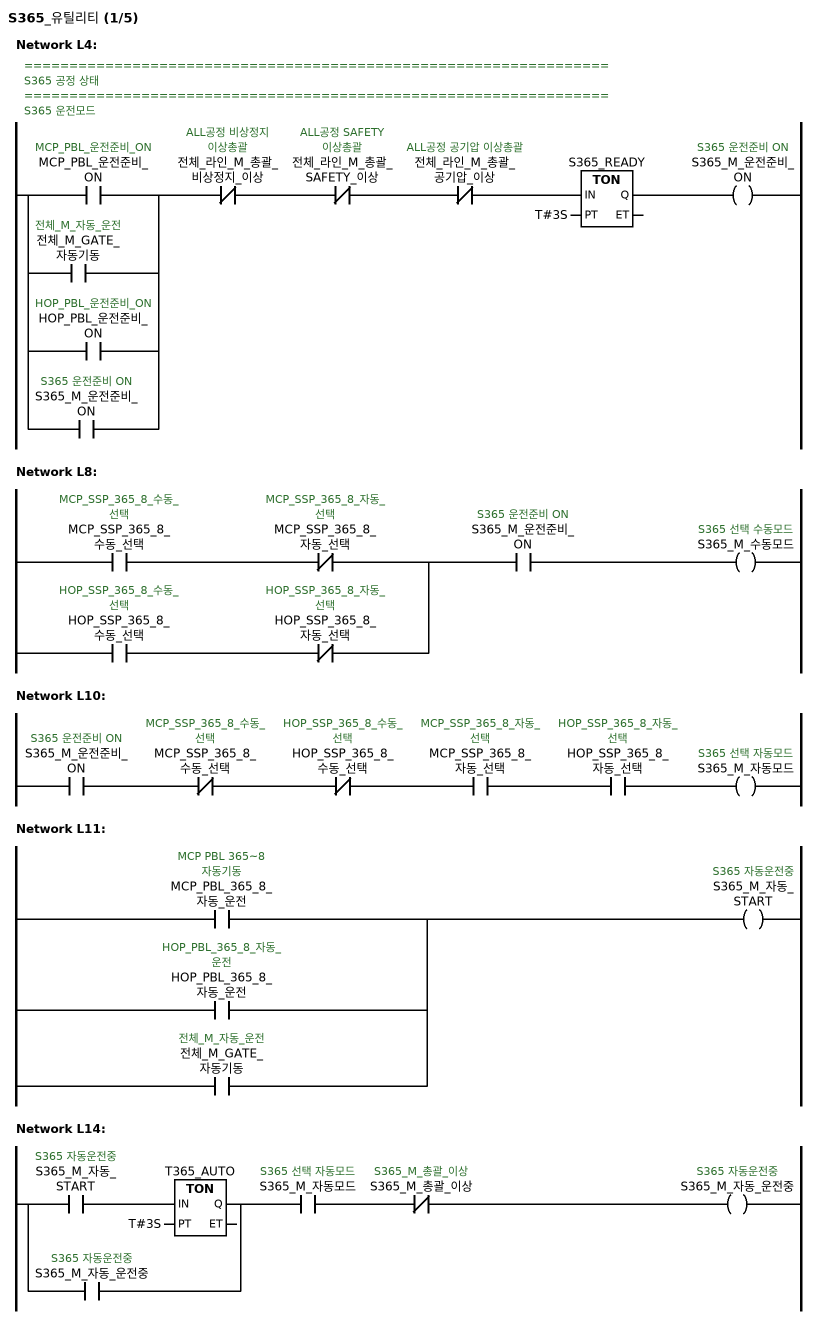
(* [picture p168: S365_유틸리티 rungs L4-L14] *)
(* ================================================================= *)
(* S365 공정 상태 *)
(* ================================================================= *)
(* S365 운전모드 *)
(* Rung L4 *)
S365_READY(IN := (MCP_PBL_운전준비_ON OR 전체_M_GATE_자동기동 OR HOP_PBL_운전준비_ON OR S365_M_운전준비_ON) AND NOT 전체_라인_M_총괄_비상정지_이상 AND NOT 전체_라인_M_총괄_SAFETY_이상 AND NOT 전체_라인_M_총괄_공기압_이상, PT := T#3S);
S365_M_운전준비_ON := S365_READY.Q;
(* Rung L8 *)
S365_M_수동모드 := ((MCP_SSP_365_8_수동_선택 AND NOT MCP_SSP_365_8_자동_선택) OR (HOP_SSP_365_8_수동_선택 AND NOT HOP_SSP_365_8_자동_선택)) AND S365_M_운전준비_ON;
(* Rung L10 *)
S365_M_자동모드 := S365_M_운전준비_ON AND NOT MCP_SSP_365_8_수동_선택 AND NOT HOP_SSP_365_8_수동_선택 AND MCP_SSP_365_8_자동_선택 AND HOP_SSP_365_8_자동_선택;
(* Rung L11 *)
S365_M_자동_START := MCP_PBL_365_8_자동_운전 OR HOP_PBL_365_8_자동_운전 OR 전체_M_GATE_자동기동;
(* Rung L14 *)
T365_AUTO(IN := S365_M_자동_START, PT := T#3S);
S365_M_자동_운전중 := (T365_AUTO.Q OR S365_M_자동_운전중) AND S365_M_자동모드 AND NOT S365_M_총괄_이상;

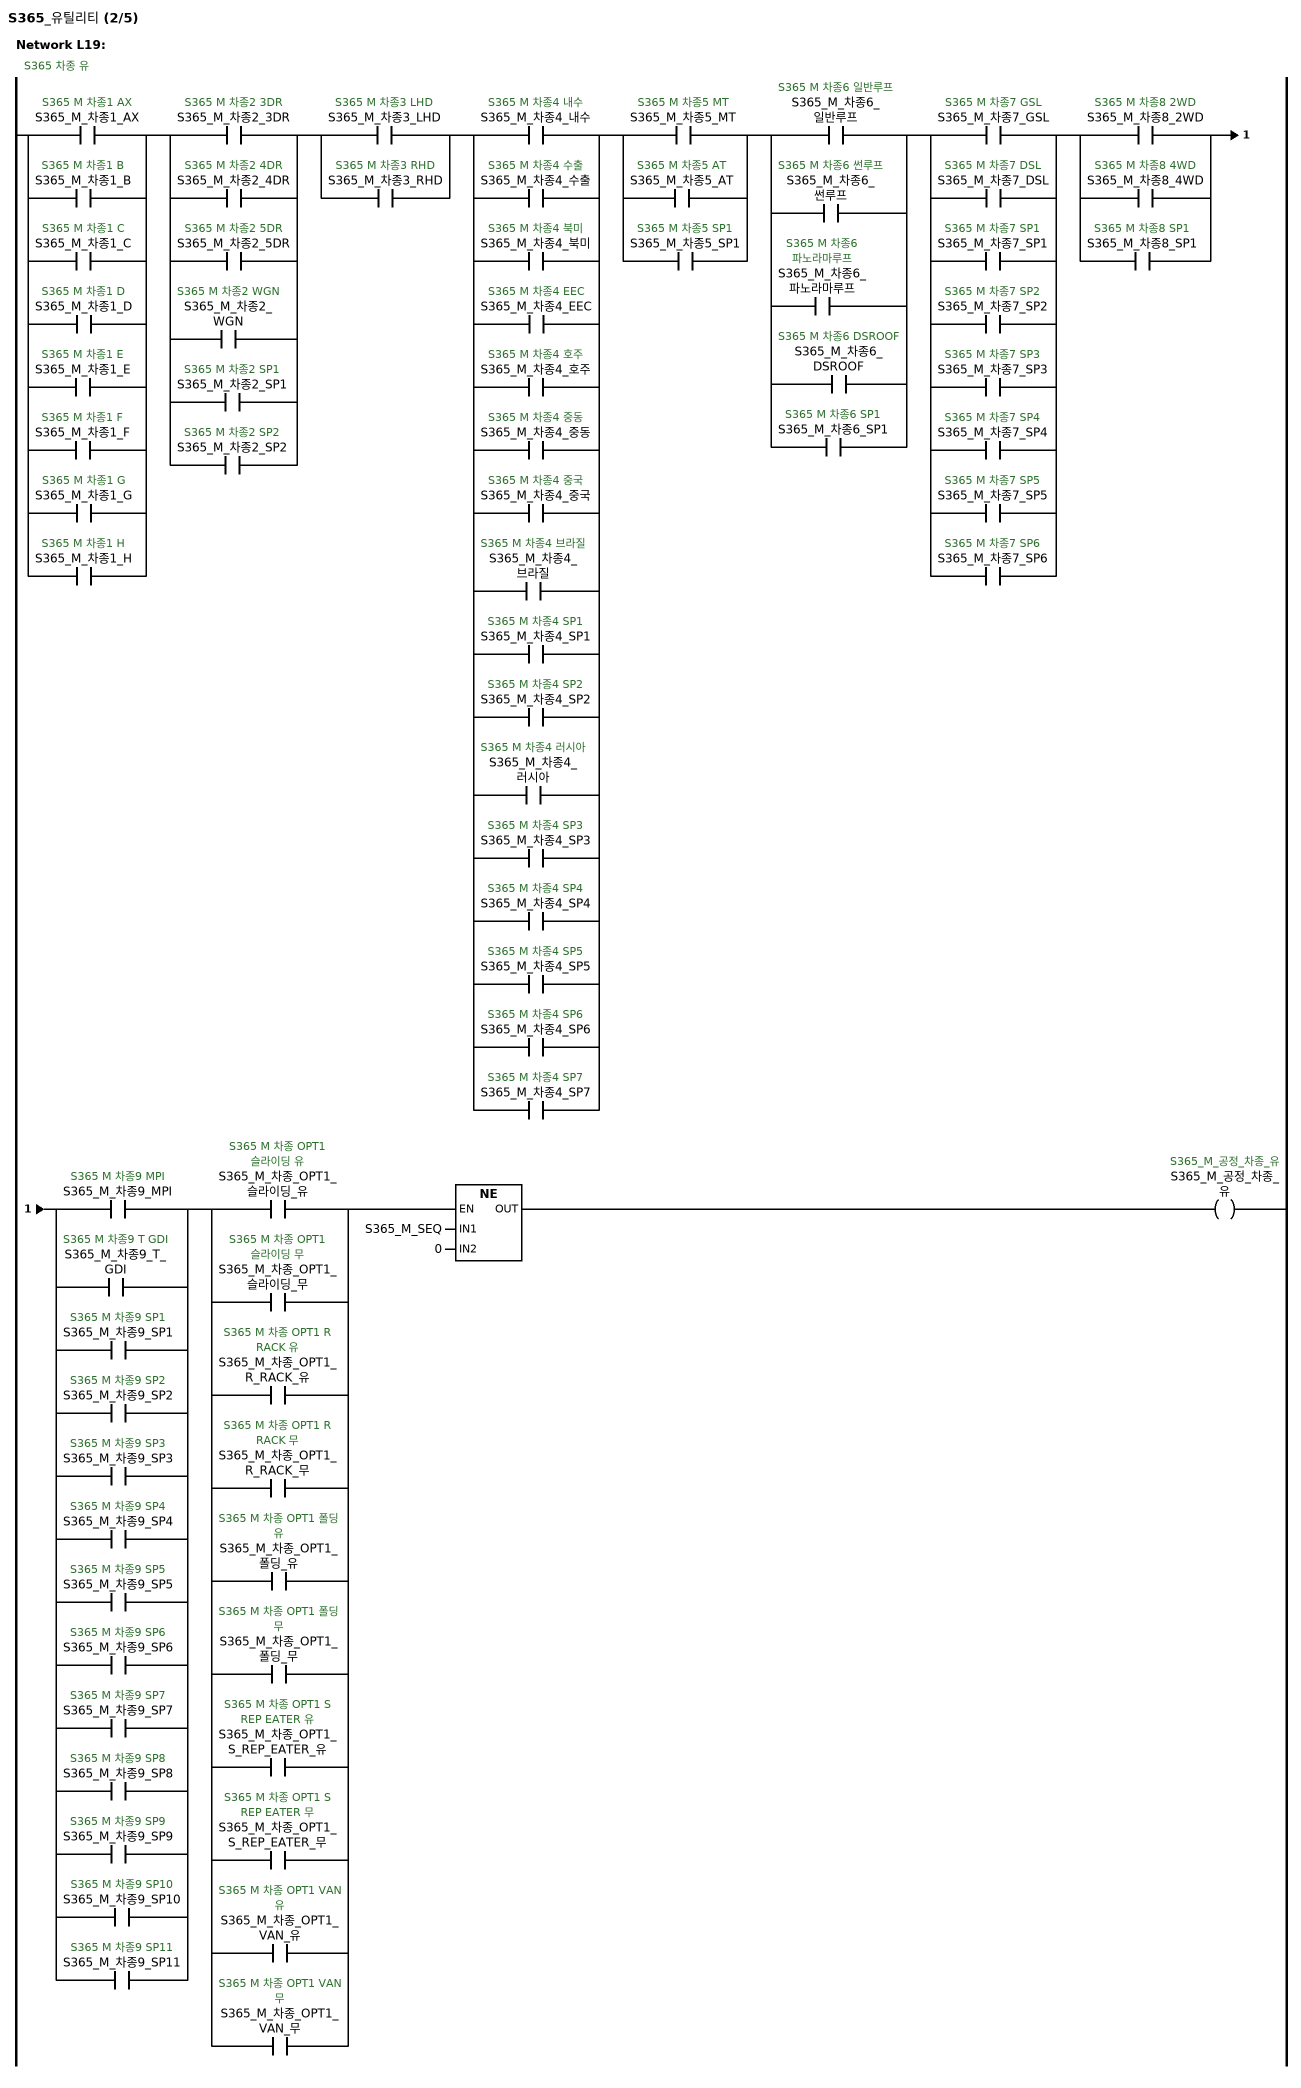
(* S365 차종 유 *)
(* Rung L19 *)
IF (S365_M_차종1_AX OR S365_M_차종1_B OR S365_M_차종1_C OR S365_M_차종1_D OR S365_M_차종1_E OR S365_M_차종1_F OR S365_M_차종1_G OR S365_M_차종1_H) AND (S365_M_차종2_3DR OR S365_M_차종2_4DR OR S365_M_차종2_5DR OR S365_M_차종2_WGN OR S365_M_차종2_SP1 OR S365_M_차종2_SP2) AND (S365_M_차종3_LHD OR S365_M_차종3_RHD) AND (S365_M_차종4_내수 OR S365_M_차종4_수출 OR S365_M_차종4_북미 OR S365_M_차종4_EEC OR S365_M_차종4_호주 OR S365_M_차종4_중동 OR S365_M_차종4_중국 OR S365_M_차종4_브라질 OR S365_M_차종4_SP1 OR S365_M_차종4_SP2 OR S365_M_차종4_러시아 OR S365_M_차종4_SP3 OR S365_M_차종4_SP4 OR S365_M_차종4_SP5 OR S365_M_차종4_SP6 OR S365_M_차종4_SP7) AND (S365_M_차종5_MT OR S365_M_차종5_AT OR S365_M_차종5_SP1) AND (S365_M_차종6_일반루프 OR S365_M_차종6_썬루프 OR S365_M_차종6_파노라마루프 OR S365_M_차종6_DSROOF OR S365_M_차종6_SP1) AND (S365_M_차종7_GSL OR S365_M_차종7_DSL OR S365_M_차종7_SP1 OR S365_M_차종7_SP2 OR S365_M_차종7_SP3 OR S365_M_차종7_SP4 OR S365_M_차종7_SP5 OR S365_M_차종7_SP6) AND (S365_M_차종8_2WD OR S365_M_차종8_4WD OR S365_M_차종8_SP1) AND (S365_M_차종9_MPI OR S365_M_차종9_T_GDI OR S365_M_차종9_SP1 OR S365_M_차종9_SP2 OR S365_M_차종9_SP3 OR S365_M_차종9_SP4 OR S365_M_차종9_SP5 OR S365_M_차종9_SP6 OR S365_M_차종9_SP7 OR S365_M_차종9_SP8 OR S365_M_차종9_SP9 OR S365_M_차종9_SP10 OR S365_M_차종9_SP11) AND (S365_M_차종_OPT1_슬라이딩_유 OR S365_M_차종_OPT1_슬라이딩_무 OR S365_M_차종_OPT1_R_RACK_유 OR S365_M_차종_OPT1_R_RACK_무 OR S365_M_차종_OPT1_폴딩_유 OR S365_M_차종_OPT1_폴딩_무 OR S365_M_차종_OPT1_S_REP_EATER_유 OR S365_M_차종_OPT1_S_REP_EATER_무 OR S365_M_차종_OPT1_VAN_유 OR S365_M_차종_OPT1_VAN_무) THEN
    _t1 := S365_M_SEQ <> 0;
END_IF;
S365_M_공정_차종_유 := _t1;

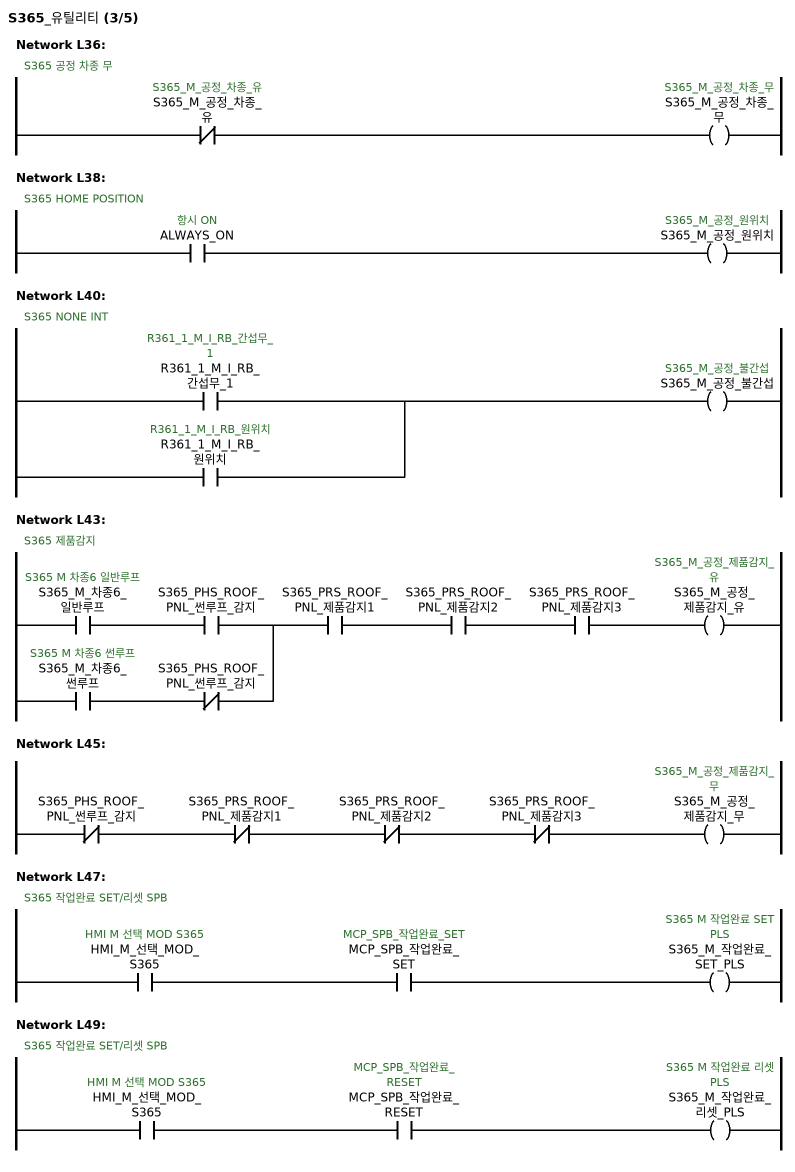
(* S365 공정 차종 무 *)
(* Rung L36 *)
S365_M_공정_차종_무 := NOT S365_M_공정_차종_유;
(* S365 HOME POSITION *)
(* Rung L38 *)
S365_M_공정_원위치 := ALWAYS_ON;
(* S365 NONE INT *)
(* Rung L40 *)
S365_M_공정_불간섭 := R361_1_M_I_RB_간섭무_1 OR R361_1_M_I_RB_원위치;
(* S365 제품감지 *)
(* Rung L43 *)
S365_M_공정_제품감지_유 := ((S365_M_차종6_일반루프 AND S365_PHS_ROOF_PNL_썬루프_감지) OR (S365_M_차종6_썬루프 AND NOT S365_PHS_ROOF_PNL_썬루프_감지)) AND S365_PRS_ROOF_PNL_제품감지1 AND S365_PRS_ROOF_PNL_제품감지2 AND S365_PRS_ROOF_PNL_제품감지3;
(* Rung L45 *)
S365_M_공정_제품감지_무 := NOT S365_PHS_ROOF_PNL_썬루프_감지 AND NOT S365_PRS_ROOF_PNL_제품감지1 AND NOT S365_PRS_ROOF_PNL_제품감지2 AND NOT S365_PRS_ROOF_PNL_제품감지3;
(* S365 작업완료 SET/리셋 SPB *)
(* Rung L47 *)
S365_M_작업완료_SET_PLS := HMI_M_선택_MOD_S365 AND MCP_SPB_작업완료_SET;
(* S365 작업완료 SET/리셋 SPB *)
(* Rung L49 *)
S365_M_작업완료_리셋_PLS := HMI_M_선택_MOD_S365 AND MCP_SPB_작업완료_RESET;

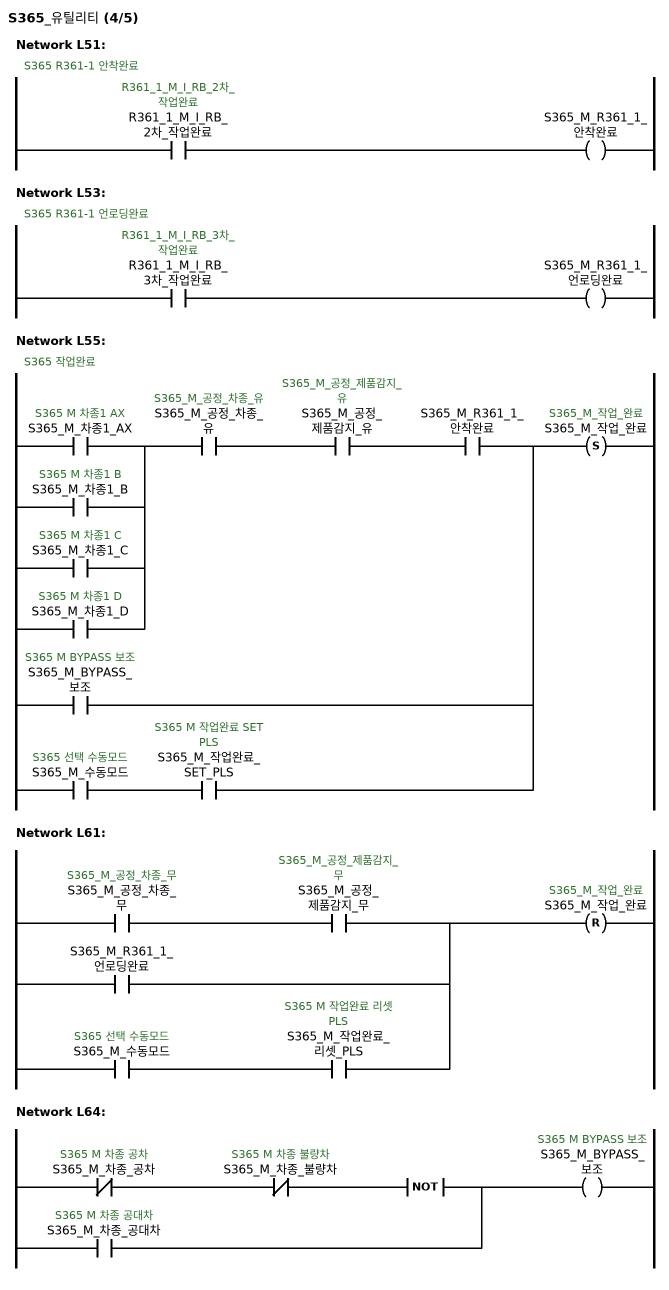
(* S365 R361-1 안착완료 *)
(* Rung L51 *)
S365_M_R361_1_안착완료 := R361_1_M_I_RB_2차_작업완료;
(* S365 R361-1 언로딩완료 *)
(* Rung L53 *)
S365_M_R361_1_언로딩완료 := R361_1_M_I_RB_3차_작업완료;
(* S365 작업완료 *)
(* Rung L55 *)
IF ((S365_M_차종1_AX OR S365_M_차종1_B OR S365_M_차종1_C OR S365_M_차종1_D) AND S365_M_공정_차종_유 AND S365_M_공정_제품감지_유 AND S365_M_R361_1_안착완료) OR S365_M_BYPASS_보조 OR (S365_M_수동모드 AND S365_M_작업완료_SET_PLS) THEN
    S365_M_작업_완료 := TRUE;
END_IF;
(* Rung L61 *)
IF (S365_M_공정_차종_무 AND S365_M_공정_제품감지_무) OR S365_M_R361_1_언로딩완료 OR (S365_M_수동모드 AND S365_M_작업완료_리셋_PLS) THEN
    S365_M_작업_완료 := FALSE;
END_IF;
(* Rung L64 *)
S365_M_BYPASS_보조 := NOT (NOT S365_M_차종_공차 AND NOT S365_M_차종_불량차) OR S365_M_차종_공대차;

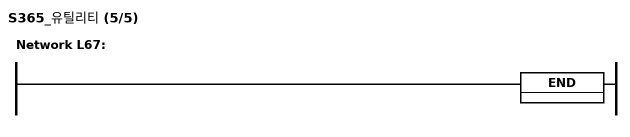
(* Rung L67 *)
END();
END_PROGRAM

PROGRAM S365_이상 (* task: 스캔 프로그램 *)
VAR
    INST10 : TON;
    INST11 : TON;
    INST12 : TON;
    INST13 : TON;
    INST14 : TON;
    INST15 : TON;
    INST16 : TON;
    INST17 : TON;
    INST18 : TON;
    INST19 : TON;
    INST20 : TON;
    INST21 : TON;
    INST22 : TON;
    INST23 : TON;
    INST24 : TON;
    INST25 : TON;
    INST8 : TON;
    INST9 : TON;
END_VAR
VAR_EXTERNAL RETAIN
    S362_M_자동_운전중 : BOOL; (* AT %MW1000.4 *) (* S362 자동운전중 *)
    S365_M_NODE_6_01_통신_이상 : BOOL; (* AT %MW2524.0 *)
    S365_M_R361_1_안착완료 : BOOL; (* AT %MW2501.1 *)
    S365_M_공정_불간섭 : BOOL; (* AT %MW2504.1 *) (* S365_M_공정_불간섭 *)
    S365_M_공정_제품감지_무 : BOOL; (* AT %MW2501.4 *) (* S365_M_공정_제품감지_무 *)
    S365_M_공정_제품감지_유 : BOOL; (* AT %MW2501.3 *) (* S365_M_공정_제품감지_유 *)
    S365_M_공정_차종_유 : BOOL; (* AT %MW2502.0 *) (* S365_M_공정_차종_유 *)
    S365_M_자동_운전중 : BOOL; (* AT %MW2500.4 *) (* S365 자동운전중 *)
    S365_M_차종6_썬루프 : BOOL; (* AT %MW10143.4 *) (* S365 M 차종6 썬루프 *)
    S365_M_차종6_일반루프 : BOOL; (* AT %MW10143.3 *) (* S365 M 차종6 일반루프 *)
    S365_M_총괄_CP_이상 : BOOL; (* AT %MW2509.7 *) (* S365 CP OFF 이상 *)
    S365_M_총괄_CT_이상 : BOOL; (* AT %MW2510.4 *) (* S365   TACK TIME 이상 *)
    S365_M_총괄_EOCR_이상 : BOOL; (* AT %MW2509.8 *) (* S365_M_총괄_EOCR_이상 *)
    S365_M_총괄_INV_이상 : BOOL; (* AT %MW2509.9 *) (* S365_M_총괄_INV_이상 *)
    S365_M_총괄_LS_이상 : BOOL; (* AT %MW2509.15 *) (* S365 LS 이상 *)
    S365_M_총괄_MATCH_이상 : BOOL; (* AT %MW2510.0 *) (* S365 매트SW 이상 *)
    S365_M_총괄_MC_이상 : BOOL; (* AT %MW2509.13 *) (* S365_M_총괄_MC_이상 *)
    S365_M_총괄_NFB_이상 : BOOL; (* AT %MW2509.11 *) (* S365_M_총괄_NFB_이상 *)
    S365_M_총괄_ROBOT_이상 : BOOL; (* AT %MW2510.1 *) (* S365 ROBOT 이상 *)
    S365_M_총괄_SAFETY_이상 : BOOL; (* AT %MW2509.2 *) (* S365 SAFETY 이상 *)
    S365_M_총괄_공기압_이상 : BOOL; (* AT %MW2509.3 *) (* S365 공기압 이상 *)
    S365_M_총괄_사양_이상 : BOOL; (* AT %MW2509.6 *) (* S365 사양 이상 *)
    S365_M_총괄_오버런_이상 : BOOL; (* AT %MW2509.12 *) (* S365_M_총괄_오버런_이상 *)
    S365_M_총괄_용접타점수_이상 : BOOL; (* AT %MW2510.2 *) (* S365 용접타점수 이상 *)
    S365_M_총괄_이상 : BOOL; (* AT %MW2509.0 *) (* S365_M_총괄_이상 *)
    S365_M_총괄_제품감지_이상 : BOOL; (* AT %MW2509.4 *) (* S365 제품감지 이상 *)
    S365_M_총괄_차종_이상 : BOOL; (* AT %MW2509.5 *) (* S365 차종 이상 *)
    S365_M_총괄_통신_이상 : BOOL; (* AT %MW2509.14 *) (* S365 통신이상 *)
    전체_M_이상_리셋 : BOOL; (* AT %MW308.2 *) (* ALL공정 PB 이상리셋 *)
END_VAR
VAR_EXTERNAL
    S365_6_1_PLC_BOX_CP_TRIP : BOOL; (* AT %MW86012.15 *) (* S365_6_1_PLC_BOX_CP_TRIP *)
    S365_PHS_ROOF_PNL_썬루프_감지 : BOOL; (* AT %MW86010.3 *)
    _0006_EB01_CFG_ER : BOOL; (* AT %MW186022.0 *) (* EB 구성 에러 *)
    _0006_EB01_DEER : BOOL; (* AT %MW186022.1 *) (* EB 운전 중 탈락 *)
    _0006_EB01_IO_DEER : BOOL; (* AT %MW186023.2 *) (* EB IO 탈락 에러 *)
    _0006_EB01_IO_TYER : BOOL; (* AT %MW186023.1 *) (* EB IO 타입 에러 *)
    _0007_EB10_CFG_ER : BOOL; (* AT %MW187040.0 *) (* EB 구성 에러 *)
    _0007_EB10_DEER : BOOL; (* AT %MW187040.1 *) (* EB 운전 중 탈락 *)
    _0007_EB10_IO_DEER : BOOL; (* AT %MW187041.2 *) (* EB IO 탈락 에러 *)
    _0007_EB10_IO_TYER : BOOL; (* AT %MW187041.1 *) (* EB IO 타입 에러 *)
END_VAR

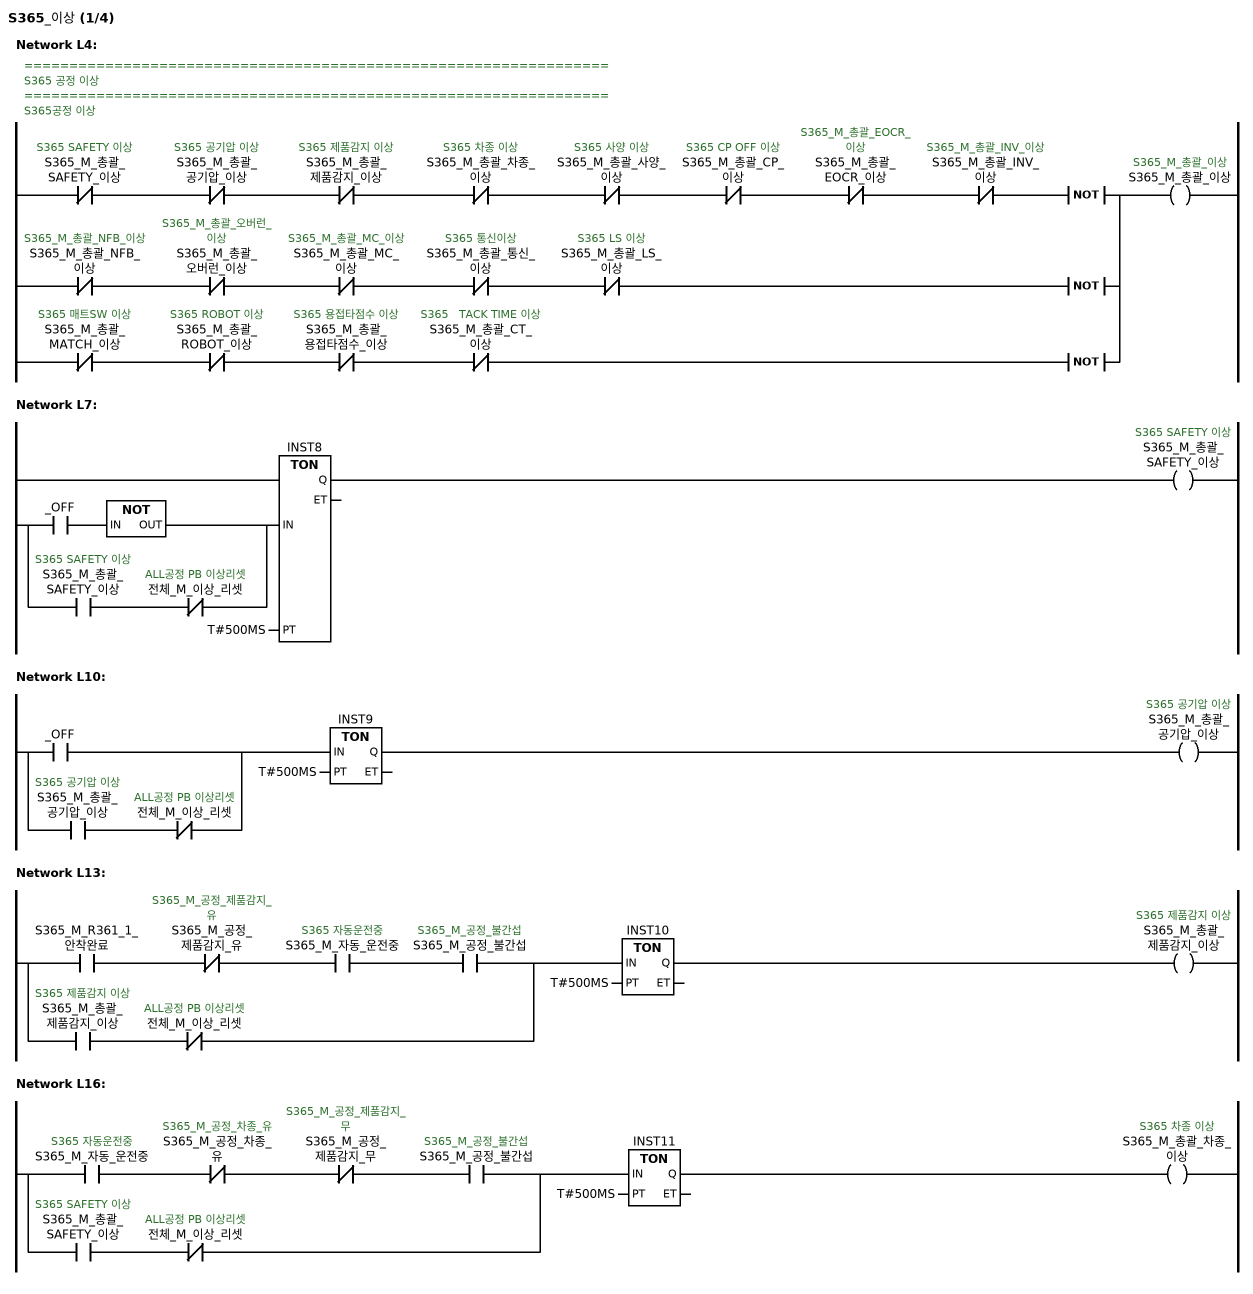
(* ================================================================= *)
(* S365 공정 이상 *)
(* ================================================================= *)
(* S365공정 이상 *)
(* Rung L4 *)
S365_M_총괄_이상 := NOT (NOT S365_M_총괄_SAFETY_이상 AND NOT S365_M_총괄_공기압_이상 AND NOT S365_M_총괄_제품감지_이상 AND NOT S365_M_총괄_차종_이상 AND NOT S365_M_총괄_사양_이상 AND NOT S365_M_총괄_CP_이상 AND NOT S365_M_총괄_EOCR_이상 AND NOT S365_M_총괄_INV_이상) OR NOT (NOT S365_M_총괄_NFB_이상 AND NOT S365_M_총괄_오버런_이상 AND NOT S365_M_총괄_MC_이상 AND NOT S365_M_총괄_통신_이상 AND NOT S365_M_총괄_LS_이상) OR NOT (NOT S365_M_총괄_MATCH_이상 AND NOT S365_M_총괄_ROBOT_이상 AND NOT S365_M_총괄_용접타점수_이상 AND NOT S365_M_총괄_CT_이상);
(* Rung L7 *)
INST8(IN := (NOT _OFF) OR (S365_M_총괄_SAFETY_이상 AND NOT 전체_M_이상_리셋), PT := T#500MS);
S365_M_총괄_SAFETY_이상 := INST8.Q;
(* Rung L10 *)
INST9(IN := _OFF OR (S365_M_총괄_공기압_이상 AND NOT 전체_M_이상_리셋), PT := T#500MS);
S365_M_총괄_공기압_이상 := INST9.Q;
(* Rung L13 *)
INST10(IN := (S365_M_R361_1_안착완료 AND NOT S365_M_공정_제품감지_유 AND S365_M_자동_운전중 AND S365_M_공정_불간섭) OR (S365_M_총괄_제품감지_이상 AND NOT 전체_M_이상_리셋), PT := T#500MS);
S365_M_총괄_제품감지_이상 := INST10.Q;
(* Rung L16 *)
INST11(IN := (S365_M_자동_운전중 AND NOT S365_M_공정_차종_유 AND NOT S365_M_공정_제품감지_무 AND S365_M_공정_불간섭) OR (S365_M_총괄_SAFETY_이상 AND NOT 전체_M_이상_리셋), PT := T#500MS);
S365_M_총괄_차종_이상 := INST11.Q;

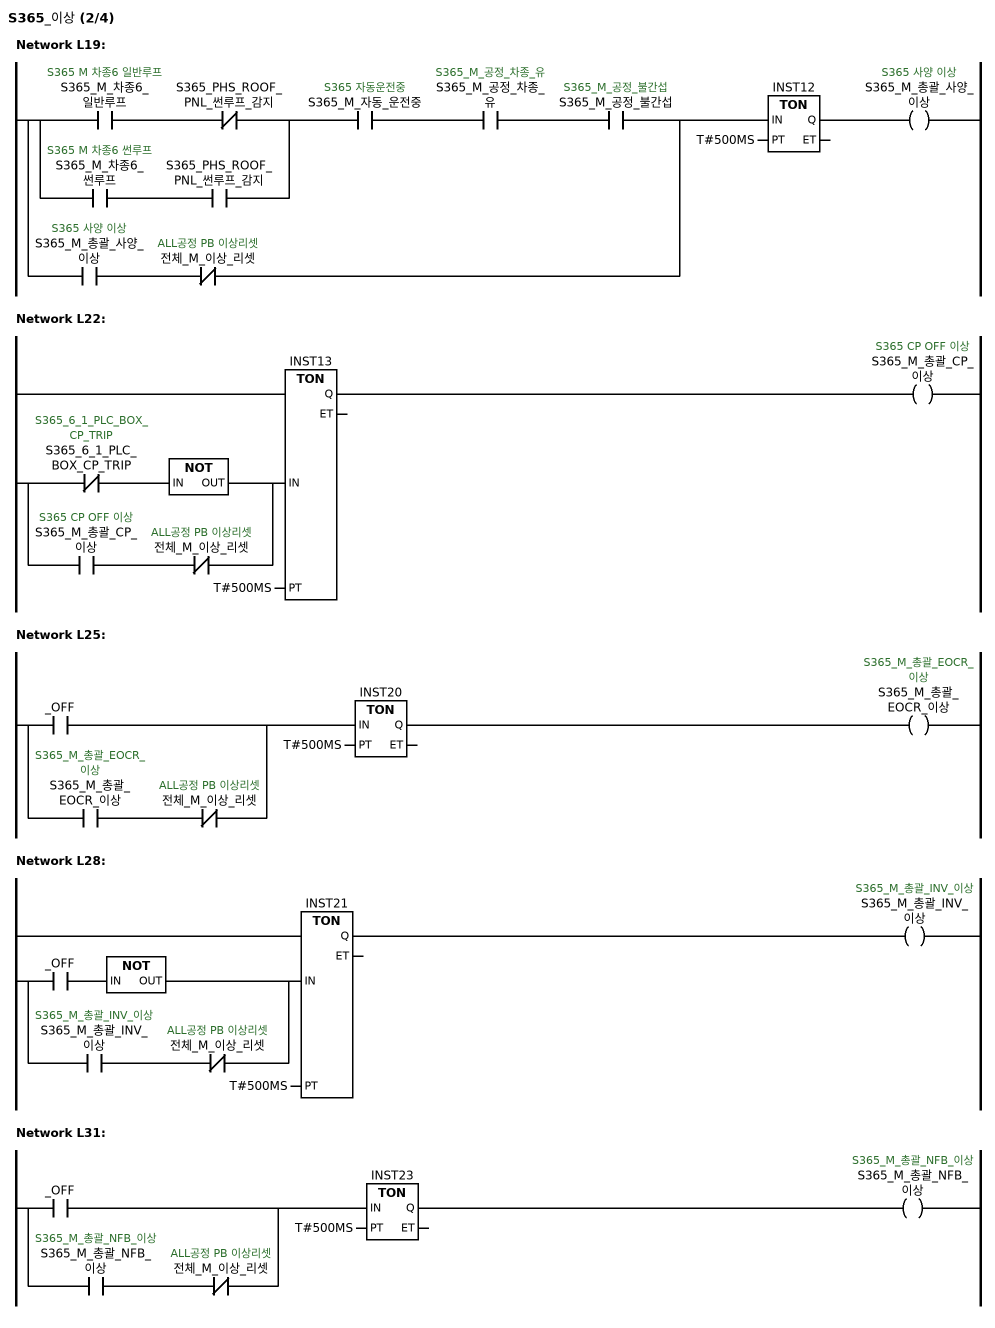
(* Rung L19 *)
INST12(IN := (((S365_M_차종6_일반루프 AND NOT S365_PHS_ROOF_PNL_썬루프_감지) OR (S365_M_차종6_썬루프 AND S365_PHS_ROOF_PNL_썬루프_감지)) AND S365_M_자동_운전중 AND S365_M_공정_차종_유 AND S365_M_공정_불간섭) OR (S365_M_총괄_사양_이상 AND NOT 전체_M_이상_리셋), PT := T#500MS);
S365_M_총괄_사양_이상 := INST12.Q;
(* Rung L22 *)
INST13(IN := (NOT (NOT S365_6_1_PLC_BOX_CP_TRIP)) OR (S365_M_총괄_CP_이상 AND NOT 전체_M_이상_리셋), PT := T#500MS);
S365_M_총괄_CP_이상 := INST13.Q;
(* Rung L25 *)
INST20(IN := _OFF OR (S365_M_총괄_EOCR_이상 AND NOT 전체_M_이상_리셋), PT := T#500MS);
S365_M_총괄_EOCR_이상 := INST20.Q;
(* Rung L28 *)
INST21(IN := (NOT _OFF) OR (S365_M_총괄_INV_이상 AND NOT 전체_M_이상_리셋), PT := T#500MS);
S365_M_총괄_INV_이상 := INST21.Q;
(* Rung L31 *)
INST23(IN := _OFF OR (S365_M_총괄_NFB_이상 AND NOT 전체_M_이상_리셋), PT := T#500MS);
S365_M_총괄_NFB_이상 := INST23.Q;

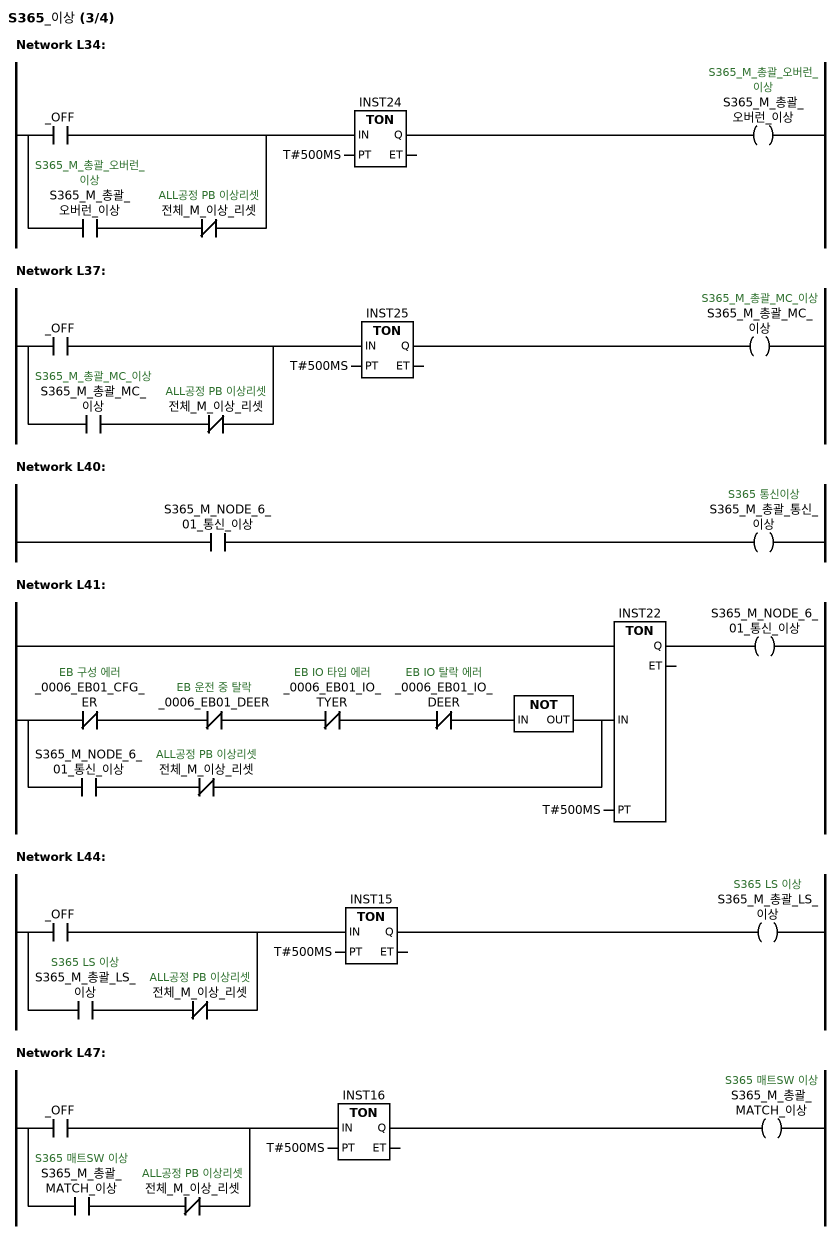
(* Rung L34 *)
INST24(IN := _OFF OR (S365_M_총괄_오버런_이상 AND NOT 전체_M_이상_리셋), PT := T#500MS);
S365_M_총괄_오버런_이상 := INST24.Q;
(* Rung L37 *)
INST25(IN := _OFF OR (S365_M_총괄_MC_이상 AND NOT 전체_M_이상_리셋), PT := T#500MS);
S365_M_총괄_MC_이상 := INST25.Q;
(* Rung L40 *)
S365_M_총괄_통신_이상 := S365_M_NODE_6_01_통신_이상;
(* Rung L41 *)
INST22(IN := (NOT (NOT _0006_EB01_CFG_ER AND NOT _0006_EB01_DEER AND NOT _0006_EB01_IO_TYER AND NOT _0006_EB01_IO_DEER)) OR (S365_M_NODE_6_01_통신_이상 AND NOT 전체_M_이상_리셋), PT := T#500MS);
S365_M_NODE_6_01_통신_이상 := INST22.Q;
(* Rung L44 *)
INST15(IN := _OFF OR (S365_M_총괄_LS_이상 AND NOT 전체_M_이상_리셋), PT := T#500MS);
S365_M_총괄_LS_이상 := INST15.Q;
(* Rung L47 *)
INST16(IN := _OFF OR (S365_M_총괄_MATCH_이상 AND NOT 전체_M_이상_리셋), PT := T#500MS);
S365_M_총괄_MATCH_이상 := INST16.Q;

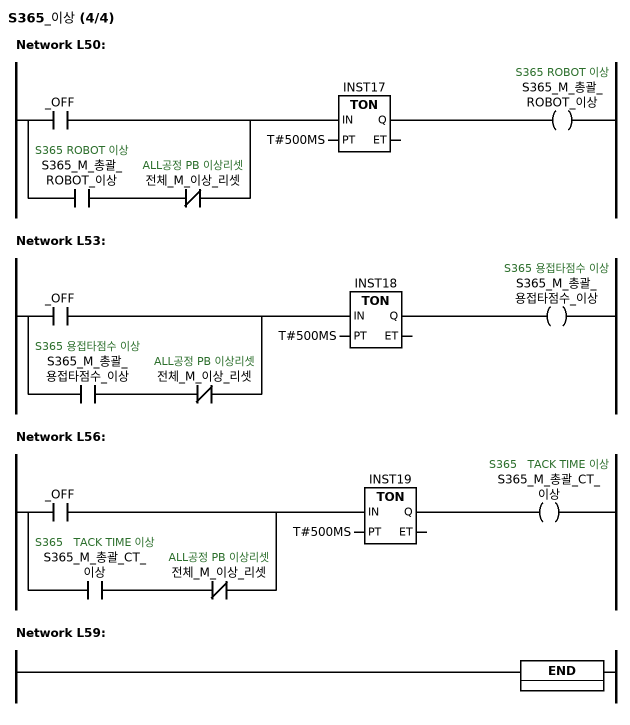
(* Rung L50 *)
INST17(IN := _OFF OR (S365_M_총괄_ROBOT_이상 AND NOT 전체_M_이상_리셋), PT := T#500MS);
S365_M_총괄_ROBOT_이상 := INST17.Q;
(* Rung L53 *)
INST18(IN := _OFF OR (S365_M_총괄_용접타점수_이상 AND NOT 전체_M_이상_리셋), PT := T#500MS);
S365_M_총괄_용접타점수_이상 := INST18.Q;
(* Rung L56 *)
INST19(IN := _OFF OR (S365_M_총괄_CT_이상 AND NOT 전체_M_이상_리셋), PT := T#500MS);
S365_M_총괄_CT_이상 := INST19.Q;
(* Rung L59 *)
END();
END_PROGRAM

PROGRAM S366_유틸리티 (* task: 스캔 프로그램 *)
VAR
    A차종 : BOOL;
    C차종 : BOOL;
    S366_READY : TON;
    T365_AUTO : TON;
    WORK_1ST : BOOL;
END_VAR
VAR_EXTERNAL
    EGIS_CWS : BOOL;
    HOP_PBL_365_8_자동_운전 : BOOL; (* AT %MW87500.7 *) (* HOP_PBL_365_8_자동_운전 *)
    HOP_PBL_운전준비_ON : BOOL; (* AT %MW87500.0 *) (* HOP_PBL_운전준비_ON *)
    HOP_SSP_365_8_수동_선택 : BOOL; (* AT %MW87500.6 *) (* HOP_SSP_365_8_수동_선택 *)
    HOP_SSP_365_8_자동_선택 : BOOL; (* AT %MW87500.5 *) (* HOP_SSP_365_8_자동_선택 *)
    MCP_PBL_365_8_자동_운전 : BOOL; (* AT %MW87630.7 *) (* MCP PBL 365~8 자동기동 *)
    MCP_PBL_운전준비_ON : BOOL; (* AT %MW87630.0 *) (* MCP_PBL_운전준비_ON *)
    MCP_SPB_작업완료_RESET : BOOL; (* AT %MW87631.6 *) (* MCP_SPB_작업완료_RESET *)
    MCP_SPB_작업완료_SET : BOOL; (* AT %MW87631.7 *) (* MCP_SPB_작업완료_SET *)
    MCP_SSP_365_8_수동_선택 : BOOL; (* AT %MW87630.5 *) (* MCP_SSP_365_8_수동_선택 *)
    MCP_SSP_365_8_자동_선택 : BOOL; (* AT %MW87630.6 *) (* MCP_SSP_365_8_자동_선택 *)
    R361_1_M_I_RB_3차_작업완료 : BOOL; (* AT %MW20011.4 *) (* R361_1_M_I_RB_3차_작업완료 *)
    R361_1_M_I_RB_4차_작업완료 : BOOL; (* AT %MW20011.5 *) (* R361_1_M_I_RB_4차_작업완료 *)
    R361_1_M_I_RB_5차_작업완료 : BOOL; (* AT %MW20011.6 *) (* R361_1_M_I_RB_5차_작업완료 *)
    R361_1_M_I_RB_간섭무_1 : BOOL; (* AT %MW20012.0 *) (* R361_1_M_I_RB_간섭무_1 *)
    R361_1_M_I_RB_원위치 : BOOL; (* AT %MW20010.3 *) (* R361_1_M_I_RB_원위치 *)
    R363_1_M_I_RB_간섭무_1 : BOOL; (* AT %MW20032.0 *) (* R363_1_M_I_RB_간섭무_1 *)
    R363_1_M_I_RB_원위치 : BOOL; (* AT %MW20030.3 *) (* R363_1_M_I_RB_원위치 *)
    R363_2_M_I_RB_2차_작업완료 : BOOL; (* AT %MW20041.3 *) (* R363_2_M_I_RB_2차_작업완료 *)
    R363_2_M_I_RB_간섭무_1 : BOOL; (* AT %MW20042.0 *) (* R363_2_M_I_RB_간섭무_1 *)
    R363_2_M_I_RB_원위치 : BOOL; (* AT %MW20040.3 *) (* R363_2_M_I_RB_원위치 *)
    R364_1_M_I_RB_1차_작업완료 : BOOL; (* AT %MW20051.2 *) (* R364_1_M_I_RB_1차_작업완료 *)
    R366_1_M_I_RB_1차_작업완료 : BOOL; (* AT %MW20061.2 *) (* R366_1_M_I_RB_1차_작업완료 *)
    R366_1_M_I_RB_3차_작업완료 : BOOL; (* AT %MW20061.4 *) (* R366_1_M_I_RB_3차_작업완료 *)
    R366_1_M_I_RB_간섭무_1 : BOOL; (* AT %MW20062.0 *) (* R366_1_M_I_RB_간섭무_1 *)
    R366_1_M_I_RB_원위치 : BOOL; (* AT %MW20060.3 *) (* R366_1_M_I_RB_원위치 *)
    S362_6_INV3_SAFETY1_ON : BOOL; (* AT %MW95015.5 *) (* S362_6_INV3_SAFETY1_ON *)
    S362_6_INV3_SAFETY2_ON : BOOL; (* AT %MW95015.6 *) (* S362_6_INV3_SAFETY2_ON *)
    S362_6_INV3_이상_리셋 : BOOL; (* AT %MW95015.3 *) (* S362_6_INV3_이상_리셋 *)
    S362_6_INV4_SAFETY1_ON : BOOL; (* AT %MW95015.13 *) (* S362_6_INV4_SAFETY1_ON *)
    S362_6_INV4_SAFETY2_ON : BOOL; (* AT %MW95015.14 *) (* S362_6_INV4_SAFETY2_ON *)
    S362_6_INV4_이상_리셋 : BOOL; (* AT %MW95015.11 *) (* S362_6_INV4_이상_리셋 *)
    S366L_PRS_AX_COM_CHECK : BOOL; (* AT %MW88100.8 *) (* S366L_PRS_AX_COM_CHECK *)
    S366L_PRS_AX_GR_CHECK : BOOL; (* AT %MW88100.9 *) (* S366L_PRS_AX_GR_CHECK *)
    S366L_PRS_AX_RAIL_CHECK : BOOL; (* AT %MW88100.11 *) (* S366L_PRS_AX_RAIL_CHECK *)
    S366L_PRS_AX_ROOF_FRT_CHECK : BOOL; (* AT %MW88100.12 *) (* S366L_PRS_AX_ROOF_FRT_CHECK *)
    S366L_PRS_AX_ROOF_RR_CHECK : BOOL; (* AT %MW88100.13 *) (* S366L_PRS_AX_ROOF_RR_CHECK *)
    S366L_PRS_AX_SR_CHECK : BOOL; (* AT %MW88100.10 *) (* S366L_PRS_AX_SR_CHECK *)
    S366R_PRS_AX_COM_CHECK : BOOL; (* AT %MW88200.8 *) (* S366R_PRS_AX_COM_CHECK *)
    S366R_PRS_AX_GR_CHECK : BOOL; (* AT %MW88200.9 *) (* S366R_PRS_AX_GR_CHECK *)
    S366R_PRS_AX_RAIL_CHECK : BOOL; (* AT %MW88200.11 *) (* S366R_PRS_AX_RAIL_CHECK *)
    S366R_PRS_AX_ROOF_FRT_CHECK : BOOL; (* AT %MW88200.12 *) (* S366R_PRS_AX_ROOF_FRT_CHECK *)
    S366R_PRS_AX_ROOF_RR_CHECK : BOOL; (* AT %MW88200.13 *) (* S366R_PRS_AX_ROOF_RR_CHECK *)
    S366R_PRS_AX_SR_CHECK : BOOL; (* AT %MW88200.10 *) (* S366R_PRS_AX_SR_CHECK *)
    S366_LS_MAINTENANCE1 : BOOL; (* AT %MW86102.0 *)
    S366_LS_MAINTENANCE2 : BOOL; (* AT %MW86102.1 *)
END_VAR
VAR_EXTERNAL RETAIN
    HMI_M_선택_MOD_S364 : BOOL; (* AT %MW6.2 *) (* HMI M 선택 MOD S364 *)
    HMI_M_선택_MOD_S366 : BOOL; (* AT %MW6.4 *) (* HMI M 선택 MOD S366 *)
    R361_1_M_SEQ : WORD; (* AT %MW10000 *) (* R361 1 M SEQ *)
    R361_1_M_차종_유 : BOOL; (* AT %MW1502.0 *)
    S362_M_총괄_이상 : BOOL; (* AT %MW1009.0 *) (* S362_M_총괄_이상 *)
    S364_M_공정_차종_무 : BOOL; (* AT %MW2002.1 *) (* S364_M_공정_차종_무 *)
    S364_M_공정_차종_유 : BOOL; (* AT %MW2002.0 *) (* S364_M_공정_차종_유 *)
    S364_M_작업완료_SET_PLS : BOOL; (* AT %MW2000.8 *) (* S364 M 작업완료 SET PLS *)
    S364_M_작업완료_리셋_PLS : BOOL; (* AT %MW2000.9 *) (* S364 M 작업완료 리셋 PLS *)
    S366_M_AX_LH_CLP_전진단 : BOOL; (* AT %MW3104.3 *) (* S366_M_AX_LH_CLP_전진단 *)
    S366_M_AX_LH_CLP_후진단 : BOOL; (* AT %MW3104.4 *) (* S366_M_AX_LH_CLP_후진단 *)
    S366_M_AX_RH_CLP_전진단 : BOOL; (* AT %MW3112.3 *) (* S366_M_AX_RH_CLP_전진단 *)
    S366_M_AX_RH_CLP_후진단 : BOOL; (* AT %MW3112.4 *) (* S366_M_AX_RH_CLP_후진단 *)
    S366_M_BYPASS_보조 : BOOL; (* AT %MW3003.15 *) (* S366 M BYPASS 보조 *)
    S366_M_LH_TURN_1_포지션단 : BOOL; (* AT %MW3101.3 *) (* S366_M_LH_TURN_1_포지션단 *)
    S366_M_LH_TURN_2_포지션단 : BOOL; (* AT %MW3101.4 *) (* S366_M_LH_TURN_2_포지션단 *)
    S366_M_LH_TURN_3_포지션단 : BOOL; (* AT %MW3101.5 *) (* S366_M_LH_TURN_3_포지션단 *)
    S366_M_LH_TURN_4_포지션단 : BOOL; (* AT %MW3101.6 *) (* S366_M_LH_TURN_4_포지션단 *)
    S366_M_R361_1_ROOF_로딩완료 : BOOL; (* AT %MW3001.2 *)
    S366_M_R361_1_동일차종_OK : BOOL; (* AT %MW3005.8 *)
    S366_M_R361_1_언로딩완료 : BOOL; (* AT %MW3001.4 *)
    S366_M_R361_1_차종매칭_조건 : BOOL; (* AT %MW3005.0 *)
    S366_M_R363_2_RAIL_로딩완료 : BOOL; (* AT %MW3001.1 *)
    S366_M_R366_1_용접가능 : BOOL; (* AT %MW3004.10 *)
    S366_M_R366_1_용접완료 : BOOL; (* AT %MW3001.3 *)
    S366_M_RAIL_로딩가능 : BOOL; (* AT %MW3004.8 *)
    S366_M_RH_TURN_1_포지션단 : BOOL; (* AT %MW3109.3 *) (* S366_M_RH_TURN_1_포지션단 *)
    S366_M_RH_TURN_2_포지션단 : BOOL; (* AT %MW3109.4 *) (* S366_M_RH_TURN_2_포지션단 *)
    S366_M_RH_TURN_3_포지션단 : BOOL; (* AT %MW3109.5 *) (* S366_M_RH_TURN_3_포지션단 *)
    S366_M_RH_TURN_4_포지션단 : BOOL; (* AT %MW3109.6 *) (* S366_M_RH_TURN_4_포지션단 *)
    S366_M_ROOF_로딩가능 : BOOL; (* AT %MW3004.9 *)
    S366_M_SAFETY_불간섭 : BOOL; (* AT %MW3004.4 *) (* S366_M_SAFETY_불간섭 *)
    S366_M_SEQ : WORD; (* AT %MW10160 *) (* S366 M SEQ *)
    S366_M_TURN_LOCK_전진단 : BOOL; (* AT %MW3100.3 *) (* S366_M_TURN_LOCK_전진단 *)
    S366_M_TURN_LOCK_후진단 : BOOL; (* AT %MW3100.4 *) (* S366_M_TURN_LOCK_후진단 *)
    S366_M_공정_AX_FRT_PNL_제품감지_이상 : BOOL; (* AT %MW3014.4 *)
    S366_M_공정_FRT_PNL_제품감지_무 : BOOL; (* AT %MW3002.13 *)
    S366_M_공정_FRT_PNL_제품감지_유 : BOOL; (* AT %MW3002.12 *)
    S366_M_공정_RAIL_제품감지_무 : BOOL; (* AT %MW3001.15 *)
    S366_M_공정_RAIL_제품감지_유 : BOOL; (* AT %MW3001.14 *)
    S366_M_공정_RR_PNL_제품감지_무 : BOOL; (* AT %MW3002.15 *)
    S366_M_공정_RR_PNL_제품감지_유 : BOOL; (* AT %MW3002.14 *)
    S366_M_공정_공용_제품감지_무 : BOOL; (* AT %MW3001.9 *)
    S366_M_공정_공용_제품감지_유 : BOOL; (* AT %MW3001.8 *)
    S366_M_공정_불간섭 : BOOL; (* AT %MW3004.1 *) (* S366_M_공정_불간섭 *)
    S366_M_공정_썬루프_제품감지_무 : BOOL; (* AT %MW3001.13 *)
    S366_M_공정_썬루프_제품감지_유 : BOOL; (* AT %MW3001.12 *)
    S366_M_공정_원위치 : BOOL; (* AT %MW3004.0 *) (* S366_M_공정_원위치 *)
    S366_M_공정_일반루프_제품감지_무 : BOOL; (* AT %MW3001.11 *)
    S366_M_공정_일반루프_제품감지_유 : BOOL; (* AT %MW3001.10 *)
    S366_M_공정_제품감지_무 : BOOL; (* AT %MW3001.7 *) (* S366_M_공정_제품감지_무 *)
    S366_M_공정_제품감지_유 : BOOL; (* AT %MW3001.6 *) (* S366_M_공정_제품감지_유 *)
    S366_M_공정_차종_무 : BOOL; (* AT %MW3002.1 *) (* S366_M_공정_차종_무 *)
    S366_M_공정_차종_유 : BOOL; (* AT %MW3002.0 *) (* S366_M_공정_차종_유 *)
    S366_M_수동모드 : BOOL; (* AT %MW3000.3 *) (* S366 선택 수동모드 *)
    S366_M_운전준비_ON : BOOL; (* AT %MW3000.0 *) (* S366 운전준비 ON *)
    S366_M_자동_START : BOOL; (* AT %MW3000.5 *) (* S366 자동운전중 *)
    S366_M_자동_운전중 : BOOL; (* AT %MW3000.4 *) (* S366 자동운전중 *)
    S366_M_자동모드 : BOOL; (* AT %MW3000.1 *) (* S366 선택 자동모드 *)
    S366_M_작업_완료 : BOOL; (* AT %MW3001.0 *) (* S366_M_작업_완료 *)
    S366_M_작업완료_SET_PLS : BOOL; (* AT %MW3000.8 *) (* S366 M 작업완료 SET PLS *)
    S366_M_작업완료_리셋_PLS : BOOL; (* AT %MW3000.9 *) (* S366 M 작업완료 리셋 PLS *)
    S366_M_차종1_AX : BOOL; (* AT %MW10161.0 *) (* S366 M 차종1 AX *)
    S366_M_차종1_B : BOOL; (* AT %MW10161.1 *) (* S366 M 차종1 B *)
    S366_M_차종1_C : BOOL; (* AT %MW10161.2 *) (* S366 M 차종1 C *)
    S366_M_차종1_D : BOOL; (* AT %MW10161.3 *) (* S366 M 차종1 D *)
    S366_M_차종1_E : BOOL; (* AT %MW10161.4 *) (* S366 M 차종1 E *)
    S366_M_차종1_F : BOOL; (* AT %MW10161.5 *) (* S366 M 차종1 F *)
    S366_M_차종1_G : BOOL; (* AT %MW10161.6 *) (* S366 M 차종1 G *)
    S366_M_차종1_H : BOOL; (* AT %MW10161.7 *) (* S366 M 차종1 H *)
    S366_M_차종2_3DR : BOOL; (* AT %MW10161.8 *) (* S366 M 차종2 3DR *)
    S366_M_차종2_4DR : BOOL; (* AT %MW10161.9 *) (* S366 M 차종2 4DR *)
    S366_M_차종2_5DR : BOOL; (* AT %MW10161.10 *) (* S366 M 차종2 5DR *)
    S366_M_차종2_SP1 : BOOL; (* AT %MW10161.12 *) (* S366 M 차종2 SP1 *)
    S366_M_차종2_SP2 : BOOL; (* AT %MW10161.13 *) (* S366 M 차종2 SP2 *)
    S366_M_차종2_WGN : BOOL; (* AT %MW10161.11 *) (* S366 M 차종2 WGN *)
    S366_M_차종3_LHD : BOOL; (* AT %MW10161.14 *) (* S366 M 차종3 LHD *)
    S366_M_차종3_RHD : BOOL; (* AT %MW10161.15 *) (* S366 M 차종3 RHD *)
    S366_M_차종4_EEC : BOOL; (* AT %MW10162.3 *) (* S366 M 차종4 EEC *)
    S366_M_차종4_SP1 : BOOL; (* AT %MW10162.8 *) (* S366 M 차종4 SP1 *)
    S366_M_차종4_SP2 : BOOL; (* AT %MW10162.9 *) (* S366 M 차종4 SP2 *)
    S366_M_차종4_SP3 : BOOL; (* AT %MW10162.11 *) (* S366 M 차종4 SP3 *)
    S366_M_차종4_SP4 : BOOL; (* AT %MW10162.12 *) (* S366 M 차종4 SP4 *)
    S366_M_차종4_SP5 : BOOL; (* AT %MW10162.13 *) (* S366 M 차종4 SP5 *)
    S366_M_차종4_SP6 : BOOL; (* AT %MW10162.14 *) (* S366 M 차종4 SP6 *)
    S366_M_차종4_SP7 : BOOL; (* AT %MW10162.15 *) (* S366 M 차종4 SP7 *)
    S366_M_차종4_내수 : BOOL; (* AT %MW10162.0 *) (* S366 M 차종4 내수 *)
    S366_M_차종4_러시아 : BOOL; (* AT %MW10162.10 *) (* S366 M 차종4 러시아 *)
    S366_M_차종4_북미 : BOOL; (* AT %MW10162.2 *) (* S366 M 차종4 북미 *)
    S366_M_차종4_브라질 : BOOL; (* AT %MW10162.7 *) (* S366 M 차종4 브라질 *)
    S366_M_차종4_수출 : BOOL; (* AT %MW10162.1 *) (* S366 M 차종4 수출 *)
    S366_M_차종4_중국 : BOOL; (* AT %MW10162.6 *) (* S366 M 차종4 중국 *)
    S366_M_차종4_중동 : BOOL; (* AT %MW10162.5 *) (* S366 M 차종4 중동 *)
    S366_M_차종4_호주 : BOOL; (* AT %MW10162.4 *) (* S366 M 차종4 호주 *)
    S366_M_차종5_AT : BOOL; (* AT %MW10163.1 *) (* S366 M 차종5 AT *)
    S366_M_차종5_MT : BOOL; (* AT %MW10163.0 *) (* S366 M 차종5 MT *)
    S366_M_차종5_SP1 : BOOL; (* AT %MW10163.2 *) (* S366 M 차종5 SP1 *)
    S366_M_차종6_DSROOF : BOOL; (* AT %MW10163.6 *) (* S366 M 차종6 DSROOF *)
    S366_M_차종6_SP1 : BOOL; (* AT %MW10163.7 *) (* S366 M 차종6 SP1 *)
    S366_M_차종6_썬루프 : BOOL; (* AT %MW10163.4 *) (* S366 M 차종6 썬루프 *)
    S366_M_차종6_일반루프 : BOOL; (* AT %MW10163.3 *) (* S366 M 차종6 일반루프 *)
    S366_M_차종6_파노라마루프 : BOOL; (* AT %MW10163.5 *) (* S366 M 차종6 파노라마루프 *)
    S366_M_차종7_DSL : BOOL; (* AT %MW10163.9 *) (* S366 M 차종7 DSL *)
    S366_M_차종7_GSL : BOOL; (* AT %MW10163.8 *) (* S366 M 차종7 GSL *)
    S366_M_차종7_SP1 : BOOL; (* AT %MW10163.10 *) (* S366 M 차종7 SP1 *)
    S366_M_차종7_SP2 : BOOL; (* AT %MW10163.11 *) (* S366 M 차종7 SP2 *)
    S366_M_차종7_SP3 : BOOL; (* AT %MW10163.12 *) (* S366 M 차종7 SP3 *)
    S366_M_차종7_SP4 : BOOL; (* AT %MW10163.13 *) (* S366 M 차종7 SP4 *)
    S366_M_차종7_SP5 : BOOL; (* AT %MW10163.14 *) (* S366 M 차종7 SP5 *)
    S366_M_차종7_SP6 : BOOL; (* AT %MW10163.15 *) (* S366 M 차종7 SP6 *)
    S366_M_차종8_2WD : BOOL; (* AT %MW10164.0 *) (* S366 M 차종8 2WD *)
    S366_M_차종8_4WD : BOOL; (* AT %MW10164.1 *) (* S366 M 차종8 4WD *)
    S366_M_차종8_SP1 : BOOL; (* AT %MW10164.2 *) (* S366 M 차종8 SP1 *)
    S366_M_차종9_MPI : BOOL; (* AT %MW10164.3 *) (* S366 M 차종9 MPI *)
    S366_M_차종9_SP1 : BOOL; (* AT %MW10164.5 *) (* S366 M 차종9 SP1 *)
    S366_M_차종9_SP10 : BOOL; (* AT %MW10164.14 *) (* S366 M 차종9 SP10 *)
    S366_M_차종9_SP11 : BOOL; (* AT %MW10164.15 *) (* S366 M 차종9 SP11 *)
    S366_M_차종9_SP2 : BOOL; (* AT %MW10164.6 *) (* S366 M 차종9 SP2 *)
    S366_M_차종9_SP3 : BOOL; (* AT %MW10164.7 *) (* S366 M 차종9 SP3 *)
    S366_M_차종9_SP4 : BOOL; (* AT %MW10164.8 *) (* S366 M 차종9 SP4 *)
    S366_M_차종9_SP5 : BOOL; (* AT %MW10164.9 *) (* S366 M 차종9 SP5 *)
    S366_M_차종9_SP6 : BOOL; (* AT %MW10164.10 *) (* S366 M 차종9 SP6 *)
    S366_M_차종9_SP7 : BOOL; (* AT %MW10164.11 *) (* S366 M 차종9 SP7 *)
    S366_M_차종9_SP8 : BOOL; (* AT %MW10164.12 *) (* S366 M 차종9 SP8 *)
    S366_M_차종9_SP9 : BOOL; (* AT %MW10164.13 *) (* S366 M 차종9 SP9 *)
    S366_M_차종9_T_GDI : BOOL; (* AT %MW10164.4 *) (* S366 M 차종9 T GDI *)
    S366_M_차종_OPT1_R_RACK_무 : BOOL; (* AT %MW10165.3 *) (* S366 M 차종 OPT1 R RACK 무 *)
    S366_M_차종_OPT1_R_RACK_유 : BOOL; (* AT %MW10165.2 *) (* S366 M 차종 OPT1 R RACK 유 *)
    S366_M_차종_OPT1_S_REP_EATER_무 : BOOL; (* AT %MW10165.7 *) (* S366 M 차종 OPT1 S REP EATER 무 *)
    S366_M_차종_OPT1_S_REP_EATER_유 : BOOL; (* AT %MW10165.6 *) (* S366 M 차종 OPT1 S REP EATER 유 *)
    S366_M_차종_OPT1_VAN_무 : BOOL; (* AT %MW10165.9 *) (* S366 M 차종 OPT1 VAN 무 *)
    S366_M_차종_OPT1_VAN_유 : BOOL; (* AT %MW10165.8 *) (* S366 M 차종 OPT1 VAN 유 *)
    S366_M_차종_OPT1_슬라이딩_무 : BOOL; (* AT %MW10165.1 *) (* S366 M 차종 OPT1 슬라이딩 무 *)
    S366_M_차종_OPT1_슬라이딩_유 : BOOL; (* AT %MW10165.0 *) (* S366 M 차종 OPT1 슬라이딩 유 *)
    S366_M_차종_OPT1_폴딩_무 : BOOL; (* AT %MW10165.5 *) (* S366 M 차종 OPT1 폴딩 무 *)
    S366_M_차종_OPT1_폴딩_유 : BOOL; (* AT %MW10165.4 *) (* S366 M 차종 OPT1 폴딩 유 *)
    S366_M_차종_공대차 : BOOL; (* AT %MW10170.12 *) (* S366 M 차종 공대차 *)
    S366_M_차종_공차 : BOOL; (* AT %MW10170.10 *) (* S366 M 차종 공차 *)
    S366_M_차종_불량차 : BOOL; (* AT %MW10170.11 *) (* S366 M 차종 불량차 *)
    S366_M_총괄_이상 : BOOL; (* AT %MW3009.0 *) (* S366_M_총괄_이상 *)
    전체_M_GATE_자동기동 : BOOL; (* AT %MW308.1 *) (* 전체_M_자동_운전 *)
    전체_M_이상_리셋 : BOOL; (* AT %MW308.2 *) (* ALL공정 PB 이상리셋 *)
    전체_라인_M_총괄_SAFETY_이상 : BOOL; (* AT %MW300.2 *) (* ALL공정 SAFETY  이상총괄 *)
    전체_라인_M_총괄_공기압_이상 : BOOL; (* AT %MW300.3 *) (* ALL공정 공기압 이상총괄 *)
    전체_라인_M_총괄_비상정지_이상 : BOOL; (* AT %MW300.1 *) (* ALL공정 비상정지 이상총괄 *)
    전체_라인_M_총괄_이상 : BOOL; (* AT %MW300.0 *) (* ALL공정 총괄이상 *)
END_VAR
VAR
    _t1 : BOOL;
    _t2 : BOOL;
    _t3 : BOOL;
    _t4 : BOOL;
    _t5 : BOOL;
    _t6 : BOOL;
    _t7 : BOOL;
    _t8 : BOOL;
END_VAR

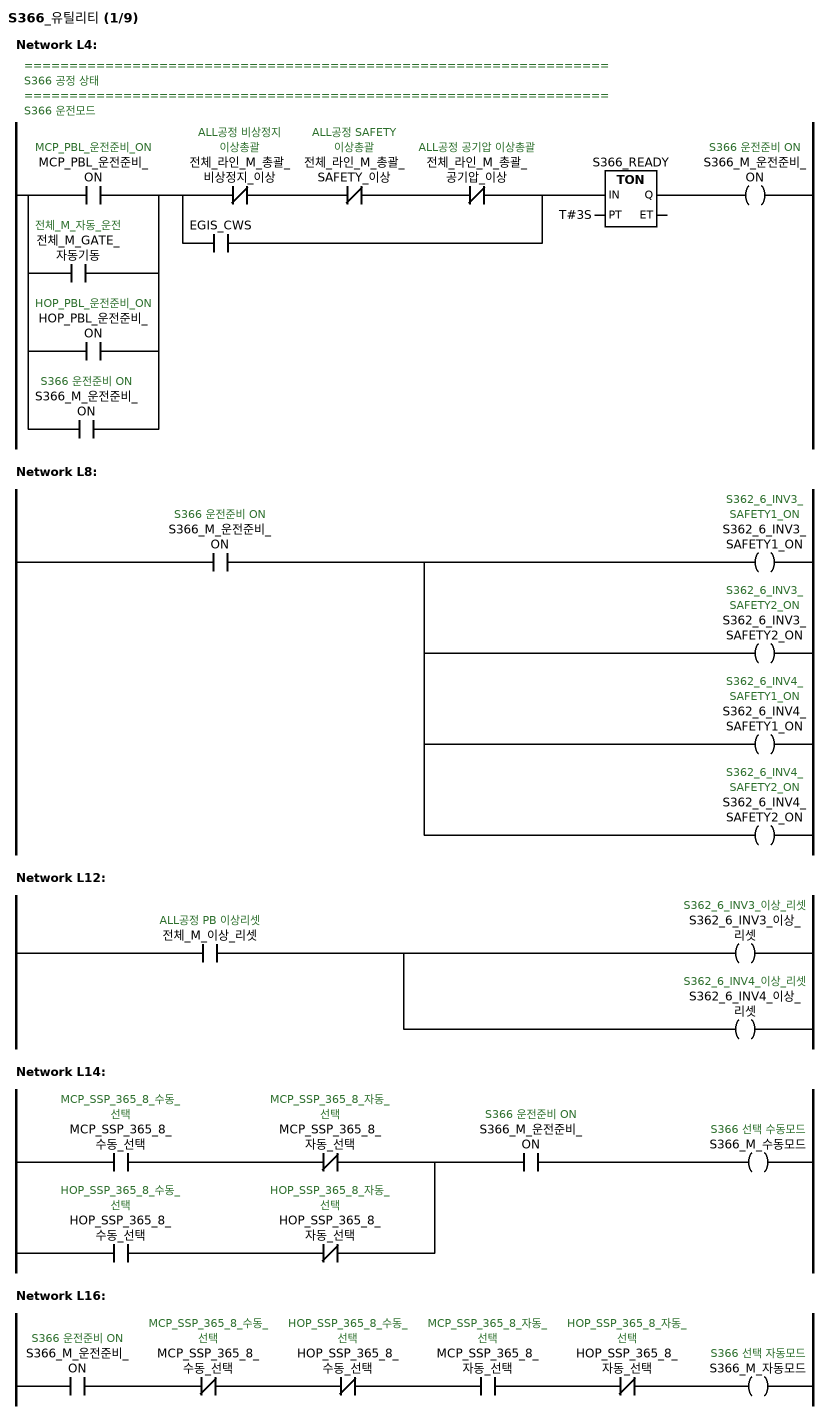
(* ================================================================= *)
(* S366 공정 상태 *)
(* ================================================================= *)
(* S366 운전모드 *)
(* Rung L4 *)
S366_READY(IN := (MCP_PBL_운전준비_ON OR 전체_M_GATE_자동기동 OR HOP_PBL_운전준비_ON OR S366_M_운전준비_ON) AND ((NOT 전체_라인_M_총괄_비상정지_이상 AND NOT 전체_라인_M_총괄_SAFETY_이상 AND NOT 전체_라인_M_총괄_공기압_이상) OR EGIS_CWS), PT := T#3S);
S366_M_운전준비_ON := S366_READY.Q;
(* Rung L8 *)
S362_6_INV3_SAFETY1_ON := S366_M_운전준비_ON;
S362_6_INV3_SAFETY2_ON := S366_M_운전준비_ON;
S362_6_INV4_SAFETY1_ON := S366_M_운전준비_ON;
S362_6_INV4_SAFETY2_ON := S366_M_운전준비_ON;
(* Rung L12 *)
S362_6_INV3_이상_리셋 := 전체_M_이상_리셋;
S362_6_INV4_이상_리셋 := 전체_M_이상_리셋;
(* Rung L14 *)
S366_M_수동모드 := ((MCP_SSP_365_8_수동_선택 AND NOT MCP_SSP_365_8_자동_선택) OR (HOP_SSP_365_8_수동_선택 AND NOT HOP_SSP_365_8_자동_선택)) AND S366_M_운전준비_ON;
(* Rung L16 *)
S366_M_자동모드 := S366_M_운전준비_ON AND NOT MCP_SSP_365_8_수동_선택 AND NOT HOP_SSP_365_8_수동_선택 AND MCP_SSP_365_8_자동_선택 AND NOT HOP_SSP_365_8_자동_선택;

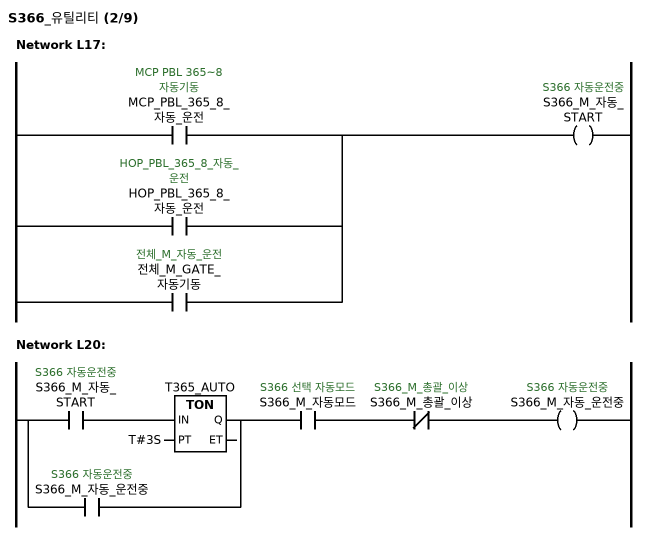
(* Rung L17 *)
S366_M_자동_START := MCP_PBL_365_8_자동_운전 OR HOP_PBL_365_8_자동_운전 OR 전체_M_GATE_자동기동;
(* Rung L20 *)
T365_AUTO(IN := S366_M_자동_START, PT := T#3S);
S366_M_자동_운전중 := (T365_AUTO.Q OR S366_M_자동_운전중) AND S366_M_자동모드 AND NOT S366_M_총괄_이상;

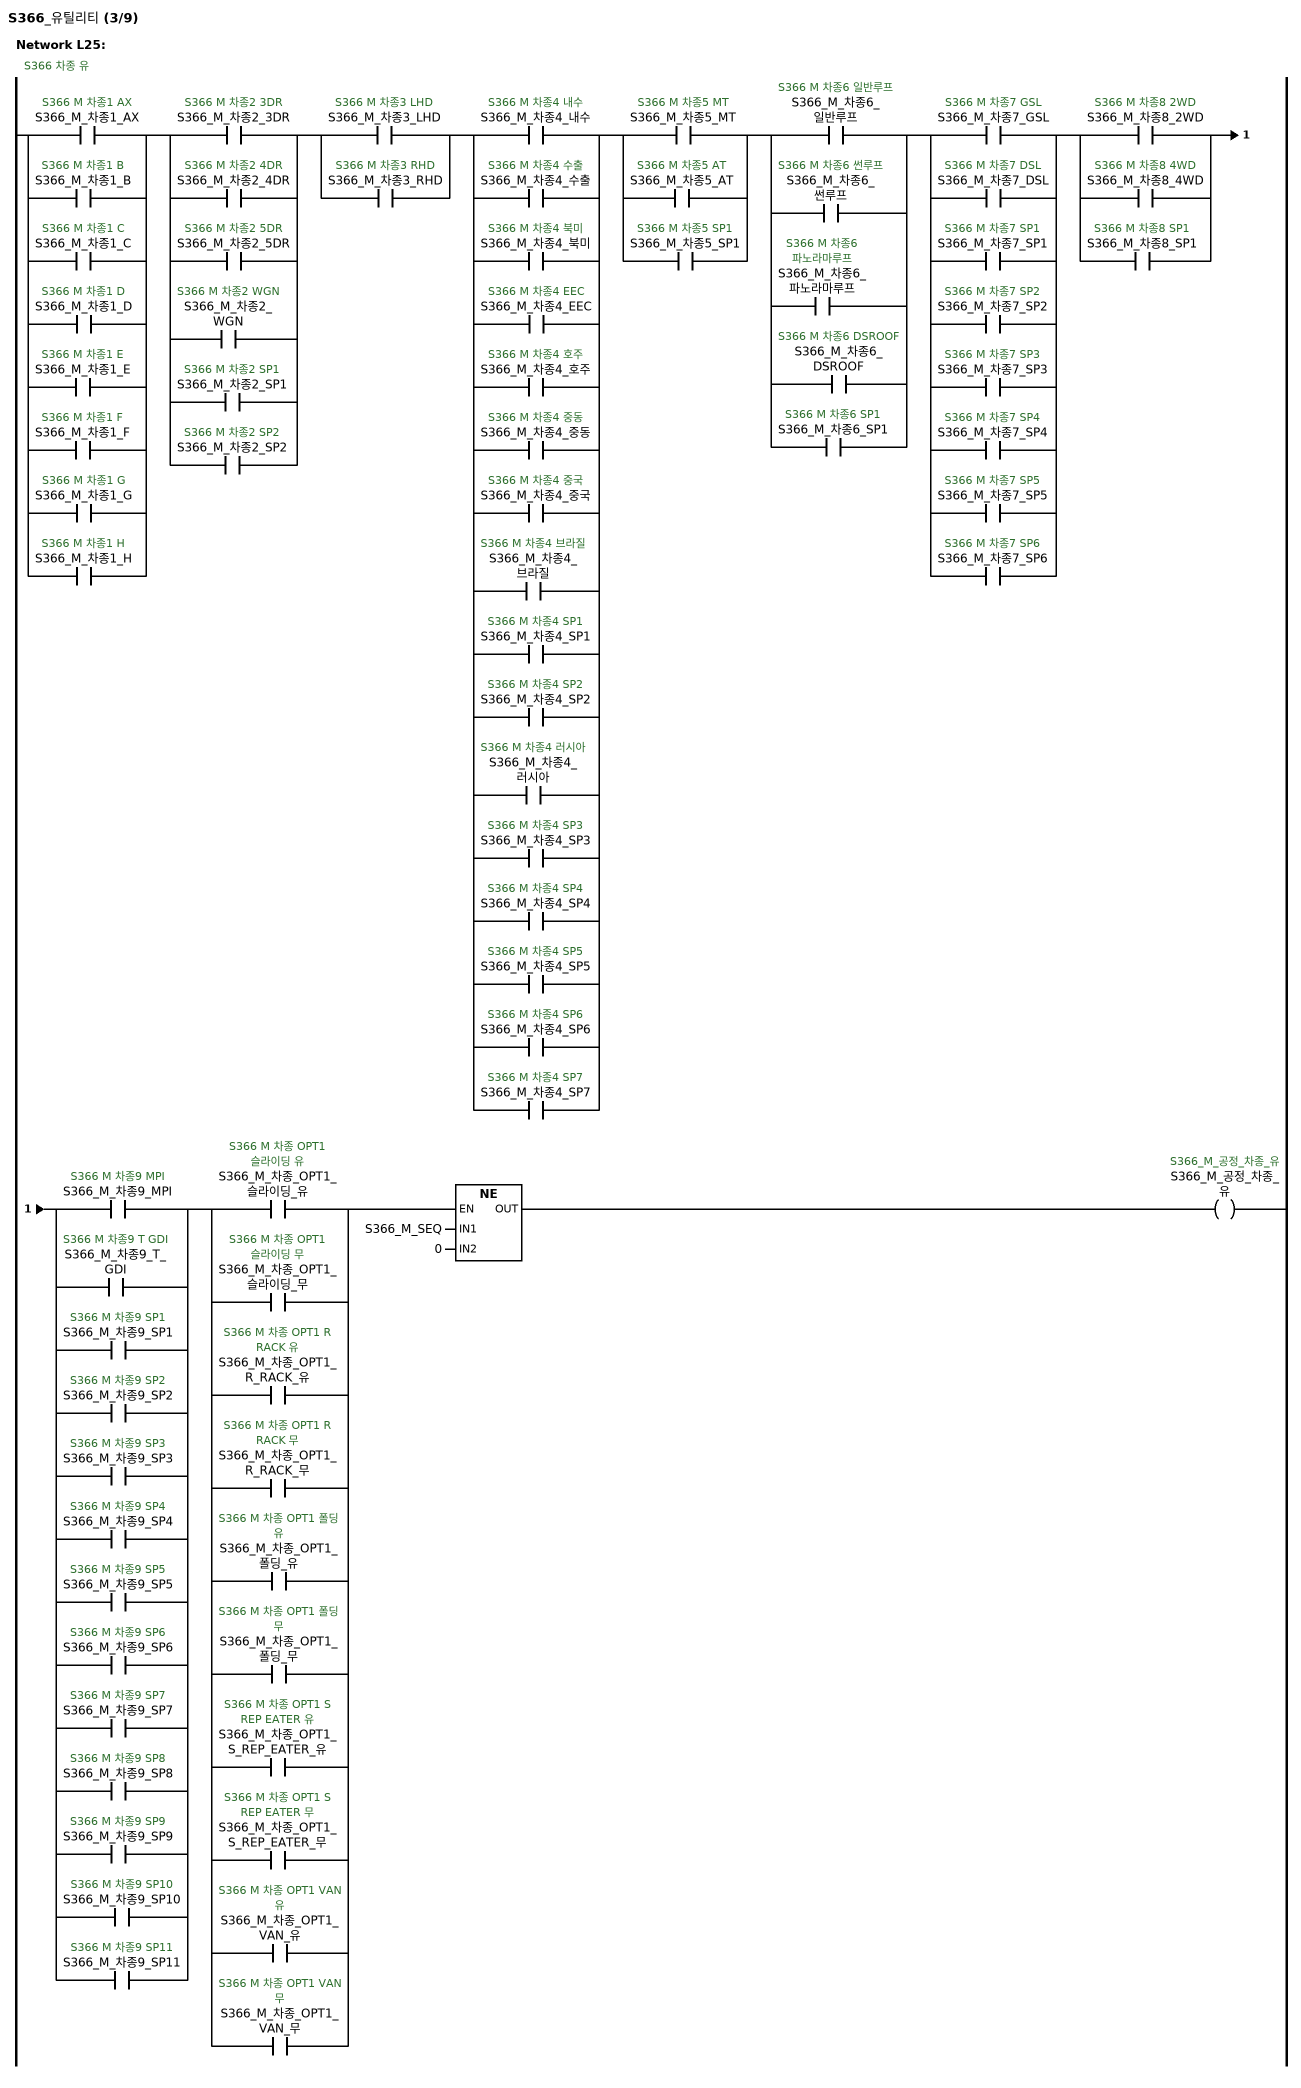
(* S366 차종 유 *)
(* Rung L25 *)
IF (S366_M_차종1_AX OR S366_M_차종1_B OR S366_M_차종1_C OR S366_M_차종1_D OR S366_M_차종1_E OR S366_M_차종1_F OR S366_M_차종1_G OR S366_M_차종1_H) AND (S366_M_차종2_3DR OR S366_M_차종2_4DR OR S366_M_차종2_5DR OR S366_M_차종2_WGN OR S366_M_차종2_SP1 OR S366_M_차종2_SP2) AND (S366_M_차종3_LHD OR S366_M_차종3_RHD) AND (S366_M_차종4_내수 OR S366_M_차종4_수출 OR S366_M_차종4_북미 OR S366_M_차종4_EEC OR S366_M_차종4_호주 OR S366_M_차종4_중동 OR S366_M_차종4_중국 OR S366_M_차종4_브라질 OR S366_M_차종4_SP1 OR S366_M_차종4_SP2 OR S366_M_차종4_러시아 OR S366_M_차종4_SP3 OR S366_M_차종4_SP4 OR S366_M_차종4_SP5 OR S366_M_차종4_SP6 OR S366_M_차종4_SP7) AND (S366_M_차종5_MT OR S366_M_차종5_AT OR S366_M_차종5_SP1) AND (S366_M_차종6_일반루프 OR S366_M_차종6_썬루프 OR S366_M_차종6_파노라마루프 OR S366_M_차종6_DSROOF OR S366_M_차종6_SP1) AND (S366_M_차종7_GSL OR S366_M_차종7_DSL OR S366_M_차종7_SP1 OR S366_M_차종7_SP2 OR S366_M_차종7_SP3 OR S366_M_차종7_SP4 OR S366_M_차종7_SP5 OR S366_M_차종7_SP6) AND (S366_M_차종8_2WD OR S366_M_차종8_4WD OR S366_M_차종8_SP1) AND (S366_M_차종9_MPI OR S366_M_차종9_T_GDI OR S366_M_차종9_SP1 OR S366_M_차종9_SP2 OR S366_M_차종9_SP3 OR S366_M_차종9_SP4 OR S366_M_차종9_SP5 OR S366_M_차종9_SP6 OR S366_M_차종9_SP7 OR S366_M_차종9_SP8 OR S366_M_차종9_SP9 OR S366_M_차종9_SP10 OR S366_M_차종9_SP11) AND (S366_M_차종_OPT1_슬라이딩_유 OR S366_M_차종_OPT1_슬라이딩_무 OR S366_M_차종_OPT1_R_RACK_유 OR S366_M_차종_OPT1_R_RACK_무 OR S366_M_차종_OPT1_폴딩_유 OR S366_M_차종_OPT1_폴딩_무 OR S366_M_차종_OPT1_S_REP_EATER_유 OR S366_M_차종_OPT1_S_REP_EATER_무 OR S366_M_차종_OPT1_VAN_유 OR S366_M_차종_OPT1_VAN_무) THEN
    _t1 := S366_M_SEQ <> 0;
END_IF;
S366_M_공정_차종_유 := _t1;

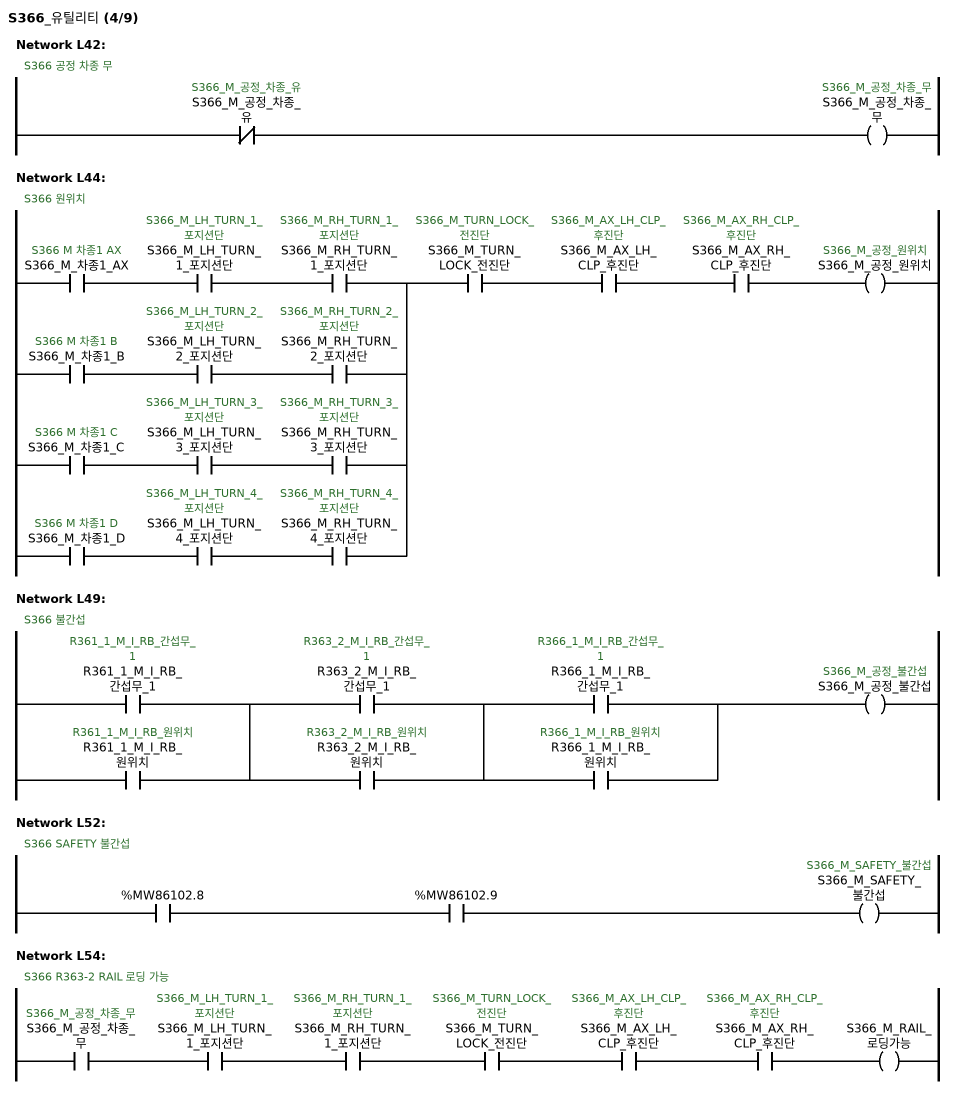
(* S366 공정 차종 무 *)
(* Rung L42 *)
S366_M_공정_차종_무 := NOT S366_M_공정_차종_유;
(* S366 원위치 *)
(* Rung L44 *)
S366_M_공정_원위치 := ((S366_M_차종1_AX AND S366_M_LH_TURN_1_포지션단 AND S366_M_RH_TURN_1_포지션단) OR (S366_M_차종1_B AND S366_M_LH_TURN_2_포지션단 AND S366_M_RH_TURN_2_포지션단) OR (S366_M_차종1_C AND S366_M_LH_TURN_3_포지션단 AND S366_M_RH_TURN_3_포지션단) OR (S366_M_차종1_D AND S366_M_LH_TURN_4_포지션단 AND S366_M_RH_TURN_4_포지션단)) AND S366_M_TURN_LOCK_전진단 AND S366_M_AX_LH_CLP_후진단 AND S366_M_AX_RH_CLP_후진단;
(* S366 불간섭 *)
(* Rung L49 *)
S366_M_공정_불간섭 := (R361_1_M_I_RB_간섭무_1 OR R361_1_M_I_RB_원위치) AND (R363_2_M_I_RB_간섭무_1 OR R363_2_M_I_RB_원위치) AND (R366_1_M_I_RB_간섭무_1 OR R366_1_M_I_RB_원위치);
(* S366 SAFETY 불간섭 *)
(* Rung L52 *)
S366_M_SAFETY_불간섭 := %MW86102.8 AND %MW86102.9;
(* S366 R363-2 RAIL 로딩 가능 *)
(* Rung L54 *)
S366_M_RAIL_로딩가능 := S366_M_공정_차종_무 AND S366_M_LH_TURN_1_포지션단 AND S366_M_RH_TURN_1_포지션단 AND S366_M_TURN_LOCK_전진단 AND S366_M_AX_LH_CLP_후진단 AND S366_M_AX_RH_CLP_후진단;

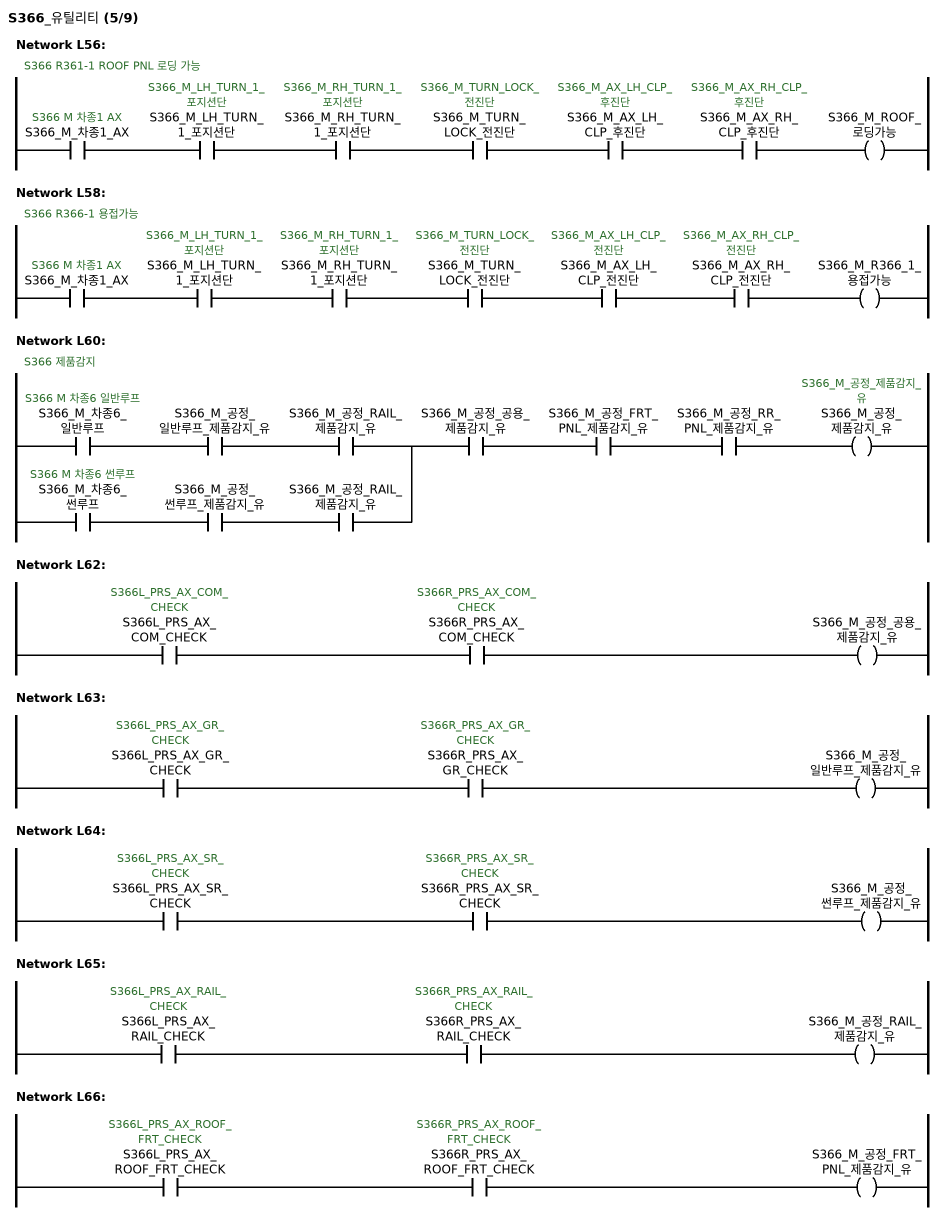
(* S366 R361-1 ROOF PNL 로딩 가능 *)
(* Rung L56 *)
S366_M_ROOF_로딩가능 := S366_M_차종1_AX AND S366_M_LH_TURN_1_포지션단 AND S366_M_RH_TURN_1_포지션단 AND S366_M_TURN_LOCK_전진단 AND S366_M_AX_LH_CLP_후진단 AND S366_M_AX_RH_CLP_후진단;
(* S366 R366-1 용접가능 *)
(* Rung L58 *)
S366_M_R366_1_용접가능 := S366_M_차종1_AX AND S366_M_LH_TURN_1_포지션단 AND S366_M_RH_TURN_1_포지션단 AND S366_M_TURN_LOCK_전진단 AND S366_M_AX_LH_CLP_전진단 AND S366_M_AX_RH_CLP_전진단;
(* S366 제품감지 *)
(* Rung L60 *)
S366_M_공정_제품감지_유 := ((S366_M_차종6_일반루프 AND S366_M_공정_일반루프_제품감지_유 AND S366_M_공정_RAIL_제품감지_유) OR (S366_M_차종6_썬루프 AND S366_M_공정_썬루프_제품감지_유 AND S366_M_공정_RAIL_제품감지_유)) AND S366_M_공정_공용_제품감지_유 AND S366_M_공정_FRT_PNL_제품감지_유 AND S366_M_공정_RR_PNL_제품감지_유;
(* Rung L62 *)
S366_M_공정_공용_제품감지_유 := S366L_PRS_AX_COM_CHECK AND S366R_PRS_AX_COM_CHECK;
(* Rung L63 *)
S366_M_공정_일반루프_제품감지_유 := S366L_PRS_AX_GR_CHECK AND S366R_PRS_AX_GR_CHECK;
(* Rung L64 *)
S366_M_공정_썬루프_제품감지_유 := S366L_PRS_AX_SR_CHECK AND S366R_PRS_AX_SR_CHECK;
(* Rung L65 *)
S366_M_공정_RAIL_제품감지_유 := S366L_PRS_AX_RAIL_CHECK AND S366R_PRS_AX_RAIL_CHECK;
(* Rung L66 *)
S366_M_공정_FRT_PNL_제품감지_유 := S366L_PRS_AX_ROOF_FRT_CHECK AND S366R_PRS_AX_ROOF_FRT_CHECK;

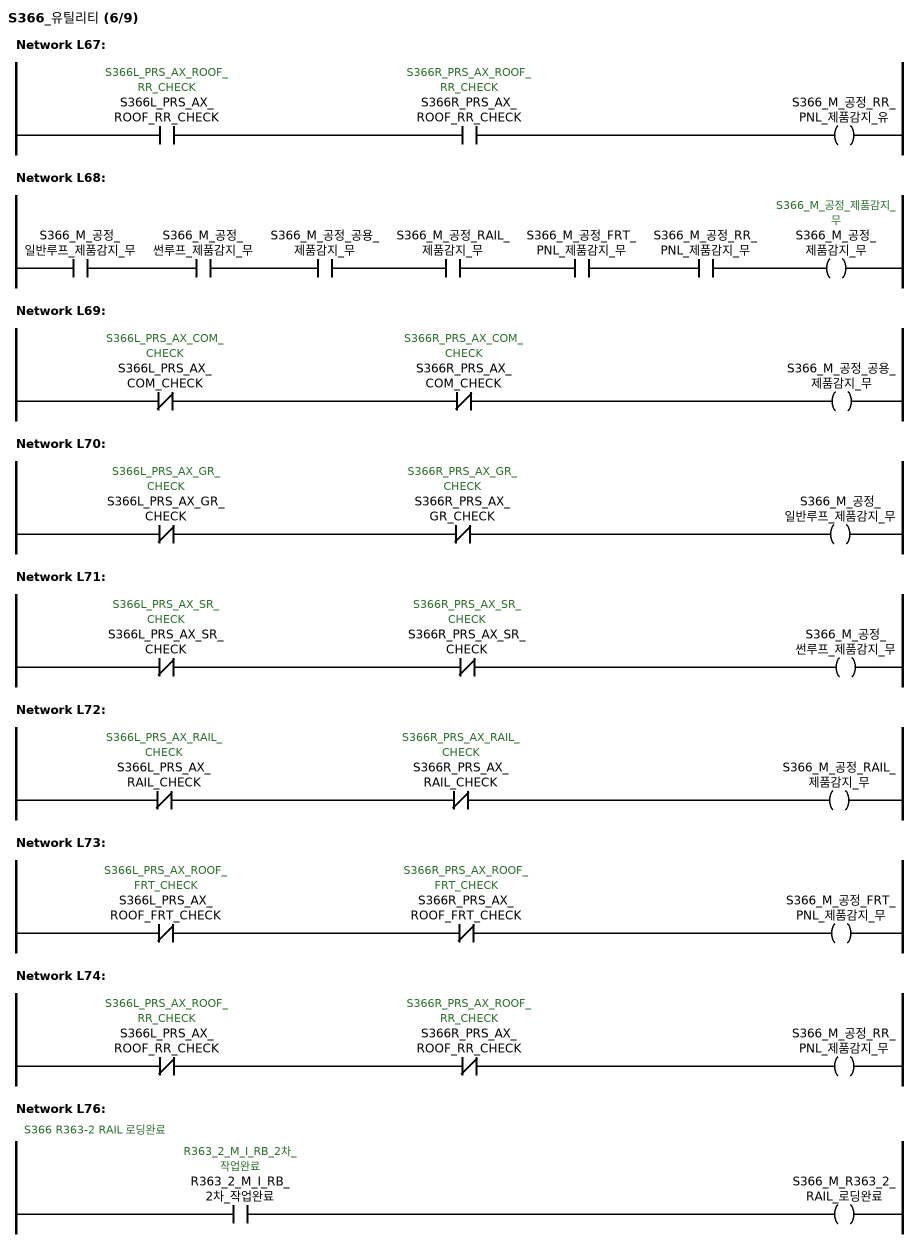
(* Rung L67 *)
S366_M_공정_RR_PNL_제품감지_유 := S366L_PRS_AX_ROOF_RR_CHECK AND S366R_PRS_AX_ROOF_RR_CHECK;
(* Rung L68 *)
S366_M_공정_제품감지_무 := S366_M_공정_일반루프_제품감지_무 AND S366_M_공정_썬루프_제품감지_무 AND S366_M_공정_공용_제품감지_무 AND S366_M_공정_RAIL_제품감지_무 AND S366_M_공정_FRT_PNL_제품감지_무 AND S366_M_공정_RR_PNL_제품감지_무;
(* Rung L69 *)
S366_M_공정_공용_제품감지_무 := NOT S366L_PRS_AX_COM_CHECK AND NOT S366R_PRS_AX_COM_CHECK;
(* Rung L70 *)
S366_M_공정_일반루프_제품감지_무 := NOT S366L_PRS_AX_GR_CHECK AND NOT S366R_PRS_AX_GR_CHECK;
(* Rung L71 *)
S366_M_공정_썬루프_제품감지_무 := NOT S366L_PRS_AX_SR_CHECK AND NOT S366R_PRS_AX_SR_CHECK;
(* Rung L72 *)
S366_M_공정_RAIL_제품감지_무 := NOT S366L_PRS_AX_RAIL_CHECK AND NOT S366R_PRS_AX_RAIL_CHECK;
(* Rung L73 *)
S366_M_공정_FRT_PNL_제품감지_무 := NOT S366L_PRS_AX_ROOF_FRT_CHECK AND NOT S366R_PRS_AX_ROOF_FRT_CHECK;
(* Rung L74 *)
S366_M_공정_RR_PNL_제품감지_무 := NOT S366L_PRS_AX_ROOF_RR_CHECK AND NOT S366R_PRS_AX_ROOF_RR_CHECK;
(* S366 R363-2 RAIL 로딩완료 *)
(* Rung L76 *)
S366_M_R363_2_RAIL_로딩완료 := R363_2_M_I_RB_2차_작업완료;

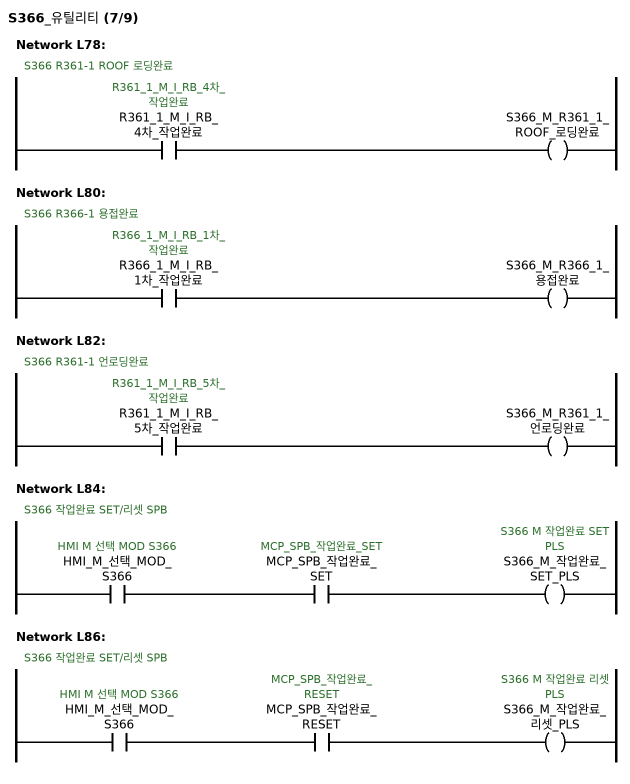
(* S366 R361-1 ROOF 로딩완료 *)
(* Rung L78 *)
S366_M_R361_1_ROOF_로딩완료 := R361_1_M_I_RB_4차_작업완료;
(* S366 R366-1 용접완료 *)
(* Rung L80 *)
S366_M_R366_1_용접완료 := R366_1_M_I_RB_1차_작업완료;
(* S366 R361-1 언로딩완료 *)
(* Rung L82 *)
S366_M_R361_1_언로딩완료 := R361_1_M_I_RB_5차_작업완료;
(* S366 작업완료 SET/리셋 SPB *)
(* Rung L84 *)
S366_M_작업완료_SET_PLS := HMI_M_선택_MOD_S366 AND MCP_SPB_작업완료_SET;
(* S366 작업완료 SET/리셋 SPB *)
(* Rung L86 *)
S366_M_작업완료_리셋_PLS := HMI_M_선택_MOD_S366 AND MCP_SPB_작업완료_RESET;

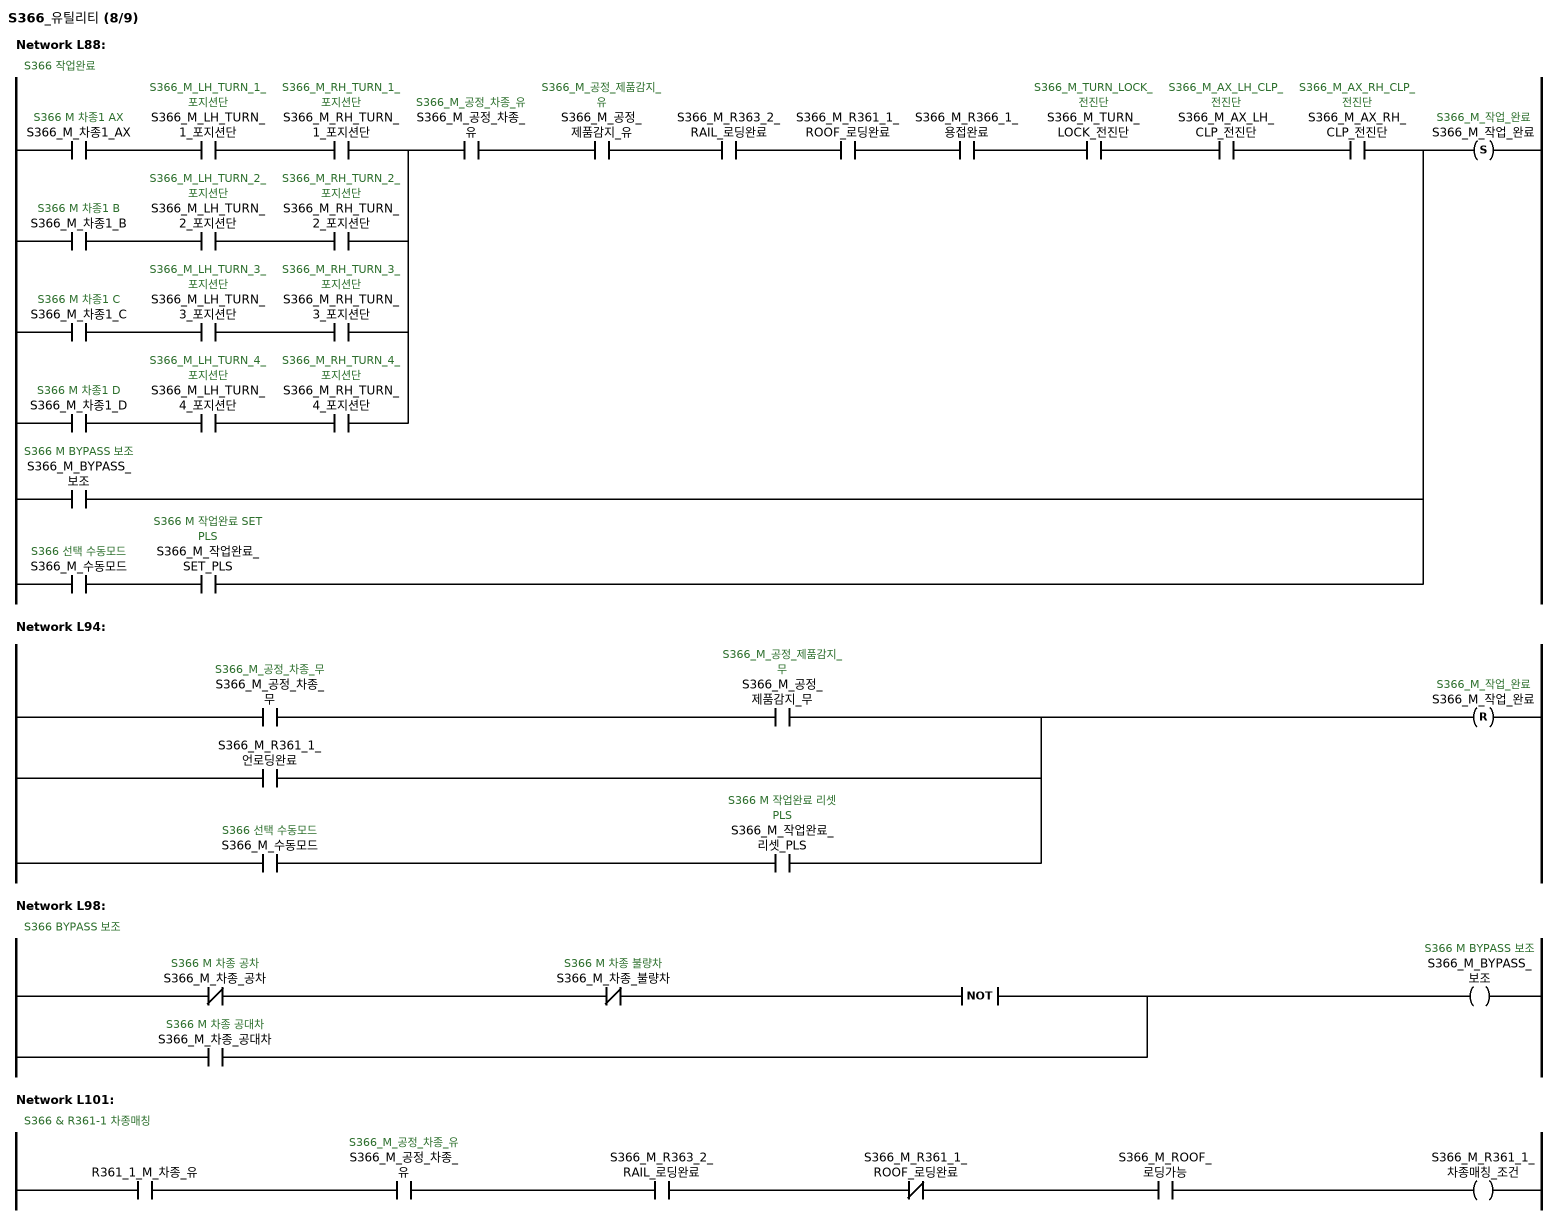
(* S366 작업완료 *)
(* Rung L88 *)
IF (((S366_M_차종1_AX AND S366_M_LH_TURN_1_포지션단 AND S366_M_RH_TURN_1_포지션단) OR (S366_M_차종1_B AND S366_M_LH_TURN_2_포지션단 AND S366_M_RH_TURN_2_포지션단) OR (S366_M_차종1_C AND S366_M_LH_TURN_3_포지션단 AND S366_M_RH_TURN_3_포지션단) OR (S366_M_차종1_D AND S366_M_LH_TURN_4_포지션단 AND S366_M_RH_TURN_4_포지션단)) AND S366_M_공정_차종_유 AND S366_M_공정_제품감지_유 AND S366_M_R363_2_RAIL_로딩완료 AND S366_M_R361_1_ROOF_로딩완료 AND S366_M_R366_1_용접완료 AND S366_M_TURN_LOCK_전진단 AND S366_M_AX_LH_CLP_전진단 AND S366_M_AX_RH_CLP_전진단) OR S366_M_BYPASS_보조 OR (S366_M_수동모드 AND S366_M_작업완료_SET_PLS) THEN
    S366_M_작업_완료 := TRUE;
END_IF;
(* Rung L94 *)
IF (S366_M_공정_차종_무 AND S366_M_공정_제품감지_무) OR S366_M_R361_1_언로딩완료 OR (S366_M_수동모드 AND S366_M_작업완료_리셋_PLS) THEN
    S366_M_작업_완료 := FALSE;
END_IF;
(* S366 BYPASS 보조 *)
(* Rung L98 *)
S366_M_BYPASS_보조 := NOT (NOT S366_M_차종_공차 AND NOT S366_M_차종_불량차) OR S366_M_차종_공대차;
(* S366 & R361-1 차종매칭 *)
(* Rung L101 *)
S366_M_R361_1_차종매칭_조건 := R361_1_M_차종_유 AND S366_M_공정_차종_유 AND S366_M_R363_2_RAIL_로딩완료 AND NOT S366_M_R361_1_ROOF_로딩완료 AND S366_M_ROOF_로딩가능;

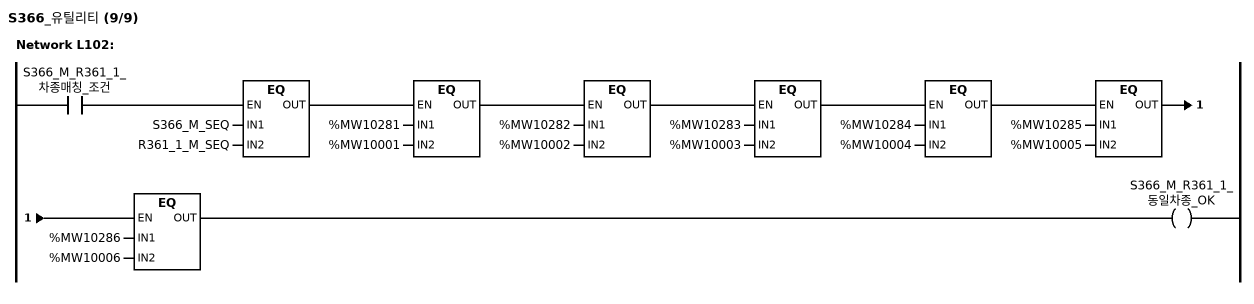
(* Rung L102 *)
IF S366_M_R361_1_차종매칭_조건 THEN _t2 := S366_M_SEQ = R361_1_M_SEQ; END_IF;
IF _t2 THEN _t3 := %MW10281 = %MW10001; END_IF;
IF _t3 THEN _t4 := %MW10282 = %MW10002; END_IF;
IF _t4 THEN _t5 := %MW10283 = %MW10003; END_IF;
IF _t5 THEN _t6 := %MW10284 = %MW10004; END_IF;
IF _t6 THEN _t7 := %MW10285 = %MW10005; END_IF;
IF _t7 THEN _t8 := %MW10286 = %MW10006; END_IF;
S366_M_R361_1_동일차종_OK := _t8;
END_PROGRAM

PROGRAM S366_동작 (* task: 스캔 프로그램 *)
VAR_EXTERNAL RETAIN
    ALWAYS_ON : BOOL; (* AT %MW3.1 *) (* 항시 ON *)
    R363_2_M_차종1_AX : BOOL; (* AT %MW10041.0 *) (* R363 2 M 차종1 AX *)
    R363_2_M_차종1_B : BOOL; (* AT %MW10041.1 *) (* R363 2 M 차종1 B *)
    R363_2_M_차종1_C : BOOL; (* AT %MW10041.2 *) (* R363 2 M 차종1 C *)
    R363_2_M_차종1_D : BOOL; (* AT %MW10041.3 *) (* R363 2 M 차종1 D *)
    S366_HOME : BOOL; (* AT %MW3048.0 *) (* S366_HOME *)
    S366_M_AX_LH_CLP_전진_LS_이상 : BOOL; (* AT %MW3104.5 *) (* S366_M_AX_LH_CLP_전진_LS_이상 *)
    S366_M_AX_LH_CLP_전진_보조 : BOOL; (* AT %MW3104.1 *) (* S366_M_AX_LH_CLP_전진_보조 *)
    S366_M_AX_LH_CLP_전진단 : BOOL; (* AT %MW3104.3 *) (* S366_M_AX_LH_CLP_전진단 *)
    S366_M_AX_LH_CLP_조건 : BOOL; (* AT %MW3104.0 *) (* S366_M_AX_LH_CLP_조건 *)
    S366_M_AX_LH_CLP_후진_LS_이상 : BOOL; (* AT %MW3104.6 *) (* S366_M_AX_LH_CLP_후진_LS_이상 *)
    S366_M_AX_LH_CLP_후진_보조 : BOOL; (* AT %MW3104.2 *) (* S366_M_AX_LH_CLP_후진_보조 *)
    S366_M_AX_LH_CLP_후진단 : BOOL; (* AT %MW3104.4 *) (* S366_M_AX_LH_CLP_후진단 *)
    S366_M_AX_RH_CLP_전진_LS_이상 : BOOL; (* AT %MW3112.5 *) (* S366_M_AX_RH_CLP_전진_LS_이상 *)
    S366_M_AX_RH_CLP_전진_보조 : BOOL; (* AT %MW3112.1 *) (* S366_M_AX_RH_CLP_전진_보조 *)
    S366_M_AX_RH_CLP_전진단 : BOOL; (* AT %MW3112.3 *) (* S366_M_AX_RH_CLP_전진단 *)
    S366_M_AX_RH_CLP_조건 : BOOL; (* AT %MW3112.0 *) (* S366_M_AX_RH_CLP_조건 *)
    S366_M_AX_RH_CLP_후진_LS_이상 : BOOL; (* AT %MW3112.6 *) (* S366_M_AX_RH_CLP_후진_LS_이상 *)
    S366_M_AX_RH_CLP_후진_보조 : BOOL; (* AT %MW3112.2 *) (* S366_M_AX_RH_CLP_후진_보조 *)
    S366_M_AX_RH_CLP_후진단 : BOOL; (* AT %MW3112.4 *) (* S366_M_AX_RH_CLP_후진단 *)
    S366_M_LH_STEP_MOVE_리셋_PLS : BOOL; (* AT %MW3101.14 *) (* S366_M_LH_STEP_MOVE_리셋_PLS *)
    S366_M_LH_TURN_1_포지션단 : BOOL; (* AT %MW3101.3 *) (* S366_M_LH_TURN_1_포지션단 *)
    S366_M_LH_TURN_2_포지션단 : BOOL; (* AT %MW3101.4 *) (* S366_M_LH_TURN_2_포지션단 *)
    S366_M_LH_TURN_3_포지션단 : BOOL; (* AT %MW3101.5 *) (* S366_M_LH_TURN_3_포지션단 *)
    S366_M_LH_TURN_4_포지션단 : BOOL; (* AT %MW3101.6 *) (* S366_M_LH_TURN_4_포지션단 *)
    S366_M_LH_TURN_MOVE_완료 : BOOL; (* AT %MW3101.8 *) (* S366_M_LH_TURN_MOVE_완료 *)
    S366_M_LH_TURN_수동_STEP_전진_보조 : BOOL; (* AT %MW3101.11 *) (* S366_M_LH_TURN_수동_STEP_전진_보조 *)
    S366_M_LH_TURN_수동_STEP_후진_보조 : BOOL; (* AT %MW3101.12 *) (* S366_M_LH_TURN_수동_STEP_후진_보조 *)
    S366_M_LH_TURN_수동_전진_보조 : BOOL; (* AT %MW3101.9 *) (* S366_M_LH_TURN_수동_전진_보조 *)
    S366_M_LH_TURN_수동_후진_보조 : BOOL; (* AT %MW3101.10 *) (* S366_M_LH_TURN_수동_후진_보조 *)
    S366_M_LH_TURN_전진_보조 : BOOL; (* AT %MW3101.1 *) (* S366_M_LH_TURN_전진_보조 *)
    S366_M_LH_TURN_조건 : BOOL; (* AT %MW3101.0 *) (* S366_M_LH_TURN_조건 *)
    S366_M_LH_TURN_후진_보조 : BOOL; (* AT %MW3101.2 *) (* S366_M_LH_TURN_후진_보조 *)
    S366_M_LH_자동_MOVE_리셋_PLS : BOOL; (* AT %MW3101.13 *) (* S366_M_LH_자동_MOVE_리셋_PLS *)
    S366_M_R361_1_ROOF_로딩완료 : BOOL; (* AT %MW3001.2 *)
    S366_M_R363_2_RAIL_로딩완료 : BOOL; (* AT %MW3001.1 *)
    S366_M_RH_STEP_MOVE_리셋_PLS : BOOL; (* AT %MW3109.14 *) (* S366_M_RH_STEP_MOVE_리셋_PLS *)
    S366_M_RH_TURN_1_포지션단 : BOOL; (* AT %MW3109.3 *) (* S366_M_RH_TURN_1_포지션단 *)
    S366_M_RH_TURN_2_포지션단 : BOOL; (* AT %MW3109.4 *) (* S366_M_RH_TURN_2_포지션단 *)
    S366_M_RH_TURN_3_포지션단 : BOOL; (* AT %MW3109.5 *) (* S366_M_RH_TURN_3_포지션단 *)
    S366_M_RH_TURN_4_포지션단 : BOOL; (* AT %MW3109.6 *) (* S366_M_RH_TURN_4_포지션단 *)
    S366_M_RH_TURN_MOVE_완료 : BOOL; (* AT %MW3109.8 *) (* S366_M_RH_TURN_MOVE_완료 *)
    S366_M_RH_TURN_수동_STEP_전진_보조 : BOOL; (* AT %MW3109.11 *) (* S366_M_RH_TURN_수동_STEP_전진_보조 *)
    S366_M_RH_TURN_수동_STEP_후진_보조 : BOOL; (* AT %MW3109.12 *) (* S366_M_RH_TURN_수동_STEP_후진_보조 *)
    S366_M_RH_TURN_수동_전진_보조 : BOOL; (* AT %MW3109.9 *) (* S366_M_RH_TURN_수동_전진_보조 *)
    S366_M_RH_TURN_수동_후진_보조 : BOOL; (* AT %MW3109.10 *) (* S366_M_RH_TURN_수동_후진_보조 *)
    S366_M_RH_TURN_전진_보조 : BOOL; (* AT %MW3109.1 *) (* S366_M_RH_TURN_전진_보조 *)
    S366_M_RH_TURN_조건 : BOOL; (* AT %MW3109.0 *) (* S366_M_RH_TURN_조건 *)
    S366_M_RH_TURN_후진_보조 : BOOL; (* AT %MW3109.2 *) (* S366_M_RH_TURN_후진_보조 *)
    S366_M_RH_자동_MOVE_리셋_PLS : BOOL; (* AT %MW3109.13 *) (* S366_M_RH_자동_MOVE_리셋_PLS *)
    S366_M_SAFETY_불간섭 : BOOL; (* AT %MW3004.4 *) (* S366_M_SAFETY_불간섭 *)
    S366_M_TURN_LOCK_전진_LS_이상 : BOOL; (* AT %MW3100.5 *) (* S366_M_TURN_LOCK_전진_LS_이상 *)
    S366_M_TURN_LOCK_전진_보조 : BOOL; (* AT %MW3100.1 *) (* S366_M_TURN_LOCK_전진_보조 *)
    S366_M_TURN_LOCK_전진단 : BOOL; (* AT %MW3100.3 *) (* S366_M_TURN_LOCK_전진단 *)
    S366_M_TURN_LOCK_조건 : BOOL; (* AT %MW3100.0 *) (* S366_M_TURN_LOCK_조건 *)
    S366_M_TURN_LOCK_후진_LS_이상 : BOOL; (* AT %MW3100.6 *) (* S366_M_TURN_LOCK_후진_LS_이상 *)
    S366_M_TURN_LOCK_후진_보조 : BOOL; (* AT %MW3100.2 *) (* S366_M_TURN_LOCK_후진_보조 *)
    S366_M_TURN_LOCK_후진단 : BOOL; (* AT %MW3100.4 *) (* S366_M_TURN_LOCK_후진단 *)
    S366_M_공정_불간섭 : BOOL; (* AT %MW3004.1 *) (* S366_M_공정_불간섭 *)
    S366_M_공정_제품감지_무 : BOOL; (* AT %MW3001.7 *) (* S366_M_공정_제품감지_무 *)
    S366_M_공정_제품감지_유 : BOOL; (* AT %MW3001.6 *) (* S366_M_공정_제품감지_유 *)
    S366_M_공정_차종_유 : BOOL; (* AT %MW3002.0 *) (* S366_M_공정_차종_유 *)
    S366_M_동작_선택_1 : BOOL; (* AT %MW3040.0 *) (* S366_M_동작_선택_1 *)
    S366_M_동작_선택_10 : BOOL; (* AT %MW3040.9 *) (* S366_M_동작_선택_10 *)
    S366_M_동작_선택_13 : BOOL; (* AT %MW3040.12 *) (* S366_M_동작_선택_13 *)
    S366_M_동작_선택_14 : BOOL; (* AT %MW3040.13 *) (* S366_M_동작_선택_14 *)
    S366_M_동작_선택_15 : BOOL; (* AT %MW3040.14 *) (* S366_M_동작_선택_15 *)
    S366_M_동작_선택_16 : BOOL; (* AT %MW3040.15 *) (* S366_M_동작_선택_16 *)
    S366_M_동작_선택_2 : BOOL; (* AT %MW3040.1 *) (* S366_M_동작_선택_2 *)
    S366_M_동작_선택_5 : BOOL; (* AT %MW3040.4 *) (* S366_M_동작_선택_5 *)
    S366_M_동작_선택_6 : BOOL; (* AT %MW3040.5 *) (* S366_M_동작_선택_6 *)
    S366_M_동작_선택_7 : BOOL; (* AT %MW3040.6 *) (* S366_M_동작_선택_7 *)
    S366_M_동작_선택_8 : BOOL; (* AT %MW3040.7 *) (* S366_M_동작_선택_8 *)
    S366_M_수동모드 : BOOL; (* AT %MW3000.3 *) (* S366 선택 수동모드 *)
    S366_M_운전준비_ON : BOOL; (* AT %MW3000.0 *) (* S366 운전준비 ON *)
    S366_M_자동_운전중 : BOOL; (* AT %MW3000.4 *) (* S366 자동운전중 *)
    S366_M_작업_완료 : BOOL; (* AT %MW3001.0 *) (* S366_M_작업_완료 *)
    S366_M_차종1_AX : BOOL; (* AT %MW10161.0 *) (* S366 M 차종1 AX *)
    S366_전진_ON : BOOL; (* AT %MW3048.1 *) (* S366_전진_ON *)
    S366_후진_ON : BOOL; (* AT %MW3048.2 *) (* S366_후진_ON *)
    전체_M_이상_리셋 : BOOL; (* AT %MW308.2 *) (* ALL공정 PB 이상리셋 *)
END_VAR
VAR
    A_차종 : BOOL;
    A차종 : BOOL;
    B_차종 : BOOL;
    C_차종 : BOOL;
    C차종 : BOOL;
    D_차종 : BOOL;
    S366_LH_AX_CLAMP : ACT_6_CYL;
    S366_RH_AX_CLAMP : ACT_6_CYL;
    S366_TURN_LOCK : ACT_6_CYL;
    T366_LH_TURN_POSI_1 : TON;
    T366_LH_TURN_POSI_2 : TON;
    T366_LH_TURN_POSI_3 : TON;
    T366_LH_TURN_POSI_4 : TON;
    T366_RH_TURN_POSI_5 : TON;
    T366_RH_TURN_POSI_6 : TON;
    T366_RH_TURN_POSI_7 : TON;
    T366_RH_TURN_POSI_8 : TON;
    WORK_1ST : BOOL;
END_VAR
VAR_EXTERNAL
    EGIS_CWS : BOOL;
    S362_6_INV3_BRAKE_CR_ON : BOOL; (* AT %MW95015.7 *) (* S362_6_INV3_BRAKE_CR_ON *)
    S362_6_INV3_RETURN : BOOL; (* AT %MW95015.1 *) (* S362_6_INV3_RETURN *)
    S362_6_INV3_TURN : BOOL; (* AT %MW95015.0 *) (* S362_6_INV3_TURN *)
    S362_6_INV4_BRAKE_CR_ON : BOOL; (* AT %MW95015.15 *) (* S362_6_INV4_BRAKE_CR_ON *)
    S362_6_INV4_RETURN : BOOL; (* AT %MW95015.9 *) (* S362_6_INV4_RETURN *)
    S362_6_INV4_TURN : BOOL; (* AT %MW95015.8 *) (* S362_6_INV4_TURN *)
    S366L_RS_AX_CLAMP_전진 : BOOL; (* AT %MW88100.0 *) (* S366L_RS_AX_CLAMP_전진 *)
    S366L_RS_AX_CLAMP_후진1 : BOOL; (* AT %MW88100.1 *) (* S366L_RS_AX_CLAMP_후진1 *)
    S366L_RS_AX_CLAMP_후진2 : BOOL; (* AT %MW88100.2 *) (* S366L_RS_AX_CLAMP_후진2 *)
    S366L_RS_AX_CLAMP_후진3 : BOOL; (* AT %MW88100.3 *) (* S366L_RS_AX_CLAMP_후진3 *)
    S366L_RS_AX_CLAMP_후진4 : BOOL; (* AT %MW88100.4 *) (* S366L_RS_AX_CLAMP_후진4 *)
    S366L_RS_AX_CLAMP_후진5 : BOOL; (* AT %MW88100.5 *) (* S366L_RS_AX_CLAMP_후진5 *)
    S366R_RS_AX_CLAMP_전진 : BOOL; (* AT %MW88200.0 *) (* S366R_RS_AX_CLAMP_전진 *)
    S366R_RS_AX_CLAMP_후진1 : BOOL; (* AT %MW88200.1 *) (* S366R_RS_AX_CLAMP_후진1 *)
    S366R_RS_AX_CLAMP_후진2 : BOOL; (* AT %MW88200.2 *) (* S366R_RS_AX_CLAMP_후진2 *)
    S366R_RS_AX_CLAMP_후진3 : BOOL; (* AT %MW88200.3 *) (* S366R_RS_AX_CLAMP_후진3 *)
    S366R_RS_AX_CLAMP_후진4 : BOOL; (* AT %MW88200.4 *) (* S366R_RS_AX_CLAMP_후진4 *)
    S366R_RS_AX_CLAMP_후진5 : BOOL; (* AT %MW88200.5 *) (* S366R_RS_AX_CLAMP_후진5 *)
    S366_INDEX_LH_TURN_감지1 : BOOL; (* AT %MW86101.4 *) (* S366_INDEX_LH_TURN_감지1 *)
    S366_INDEX_LH_TURN_감지2 : BOOL; (* AT %MW86101.5 *) (* S366_INDEX_LH_TURN_감지2 *)
    S366_INDEX_LH_TURN_감지3 : BOOL; (* AT %MW86101.6 *) (* S366_INDEX_LH_TURN_감지3 *)
    S366_INDEX_LH_TURN_원점 : BOOL; (* AT %MW86101.7 *) (* S366_INDEX_LH_TURN_원점 *)
    S366_INDEX_RH_TURN_감지1 : BOOL; (* AT %MW86101.0 *) (* S366_INDEX_RH_TURN_감지1 *)
    S366_INDEX_RH_TURN_감지2 : BOOL; (* AT %MW86101.1 *) (* S366_INDEX_RH_TURN_감지2 *)
    S366_INDEX_RH_TURN_감지3 : BOOL; (* AT %MW86101.2 *) (* S366_INDEX_RH_TURN_감지3 *)
    S366_INDEX_RH_TURN_원점 : BOOL; (* AT %MW86101.3 *) (* S366_INDEX_RH_TURN_원점 *)
    S366_M_AX_LH_CLP_전진_LAMP : WORD; (* AT %MW12608 *) (* S366_M_AX_LH_CLP_전진_LAMP *)
    S366_M_AX_LH_CLP_후진_LAMP : WORD; (* AT %MW12609 *) (* S366_M_AX_LH_CLP_후진_LAMP *)
    S366_M_AX_RH_CLP_전진_LAMP : WORD; (* AT %MW12624 *) (* S366_M_AX_RH_CLP_전진_LAMP *)
    S366_M_AX_RH_CLP_후진_LAMP : WORD; (* AT %MW12625 *) (* S366_M_AX_RH_CLP_후진_LAMP *)
    S366_M_TURN_LOCK_전진_LAMP : WORD; (* AT %MW12600 *) (* S366_M_TURN_LOCK_전진_LAMP *)
    S366_M_TURN_LOCK_후진_LAMP : WORD; (* AT %MW12601 *) (* S366_M_TURN_LOCK_후진_LAMP *)
    S366_RS_AX_IDX_LOCK_전진1 : BOOL; (* AT %MW86100.0 *) (* S366_RS_AX_IDX_LOCK_전진1 *)
    S366_RS_AX_IDX_LOCK_전진2 : BOOL; (* AT %MW86100.2 *) (* S366_RS_AX_IDX_LOCK_전진2 *)
    S366_RS_AX_IDX_LOCK_후진1 : BOOL; (* AT %MW86100.1 *) (* S366_RS_AX_IDX_LOCK_후진1 *)
    S366_RS_AX_IDX_LOCK_후진2 : BOOL; (* AT %MW86100.3 *) (* S366_RS_AX_IDX_LOCK_후진2 *)
    S366_SOL_AX_LH_CLP_전진 : BOOL; (* AT %MW98101.0 *)
    S366_SOL_AX_LH_CLP_후진 : BOOL; (* AT %MW98101.1 *)
    S366_SOL_AX_LOCK_G_전진 : BOOL; (* AT %MW96103.0 *) (* S366_SOL_AX_LOCK_G_전진 *)
    S366_SOL_AX_LOCK_G_후진 : BOOL; (* AT %MW96103.1 *) (* S366_SOL_AX_LOCK_G_후진 *)
    S366_SOL_AX_RH_CLP_전진 : BOOL; (* AT %MW98201.0 *)
    S366_SOL_AX_RH_CLP_후진 : BOOL; (* AT %MW98201.1 *)
END_VAR

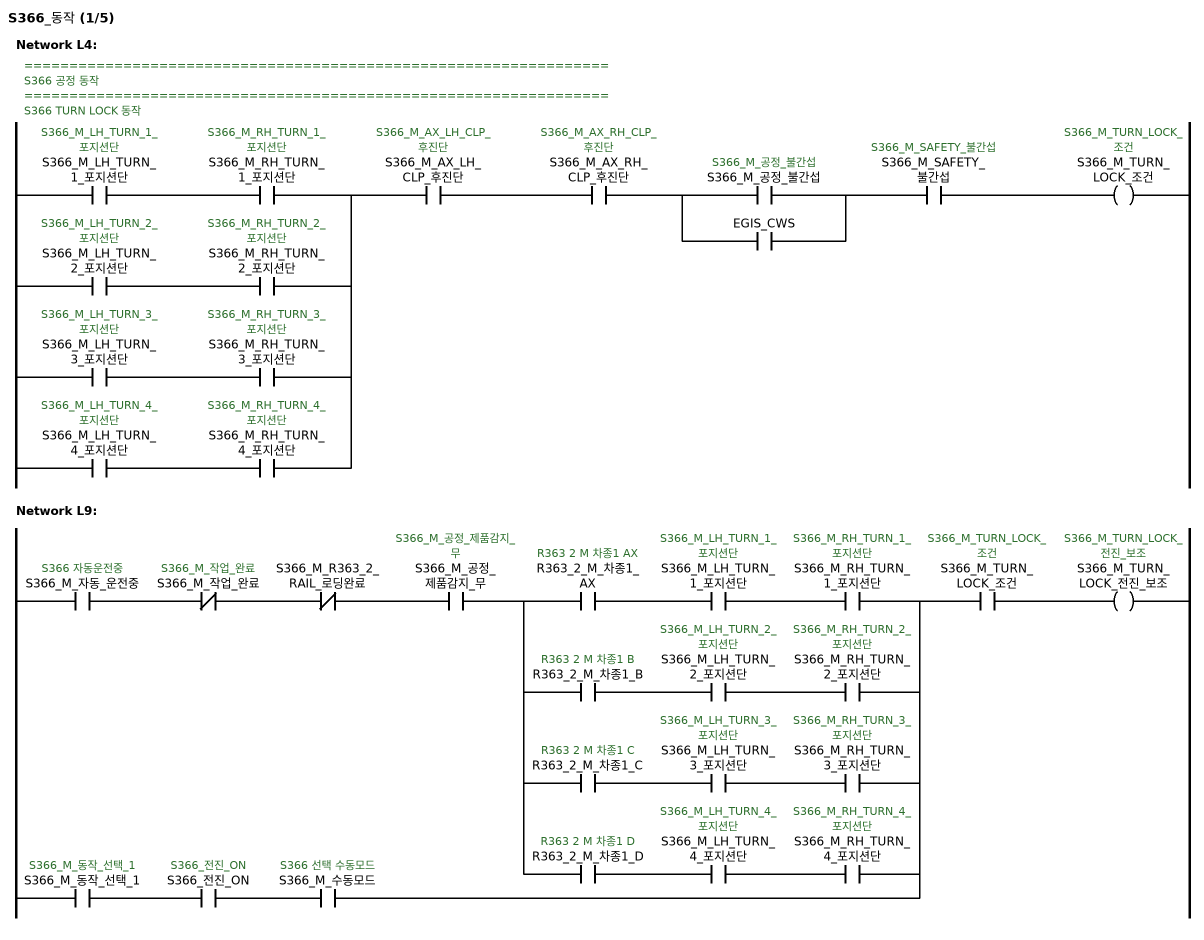
(* ================================================================= *)
(* S366 공정 동작 *)
(* ================================================================= *)
(* S366 TURN LOCK 동작 *)
(* Rung L4 *)
S366_M_TURN_LOCK_조건 := ((S366_M_LH_TURN_1_포지션단 AND S366_M_RH_TURN_1_포지션단) OR (S366_M_LH_TURN_2_포지션단 AND S366_M_RH_TURN_2_포지션단) OR (S366_M_LH_TURN_3_포지션단 AND S366_M_RH_TURN_3_포지션단) OR (S366_M_LH_TURN_4_포지션단 AND S366_M_RH_TURN_4_포지션단)) AND S366_M_AX_LH_CLP_후진단 AND S366_M_AX_RH_CLP_후진단 AND (S366_M_공정_불간섭 OR EGIS_CWS) AND S366_M_SAFETY_불간섭;
(* Rung L9 *)
S366_M_TURN_LOCK_전진_보조 := ((S366_M_자동_운전중 AND NOT S366_M_작업_완료 AND NOT S366_M_R363_2_RAIL_로딩완료 AND S366_M_공정_제품감지_무 AND ((R363_2_M_차종1_AX AND S366_M_LH_TURN_1_포지션단 AND S366_M_RH_TURN_1_포지션단) OR (R363_2_M_차종1_B AND S366_M_LH_TURN_2_포지션단 AND S366_M_RH_TURN_2_포지션단) OR (R363_2_M_차종1_C AND S366_M_LH_TURN_3_포지션단 AND S366_M_RH_TURN_3_포지션단) OR (R363_2_M_차종1_D AND S366_M_LH_TURN_4_포지션단 AND S366_M_RH_TURN_4_포지션단))) OR (S366_M_동작_선택_1 AND S366_전진_ON AND S366_M_수동모드)) AND S366_M_TURN_LOCK_조건;

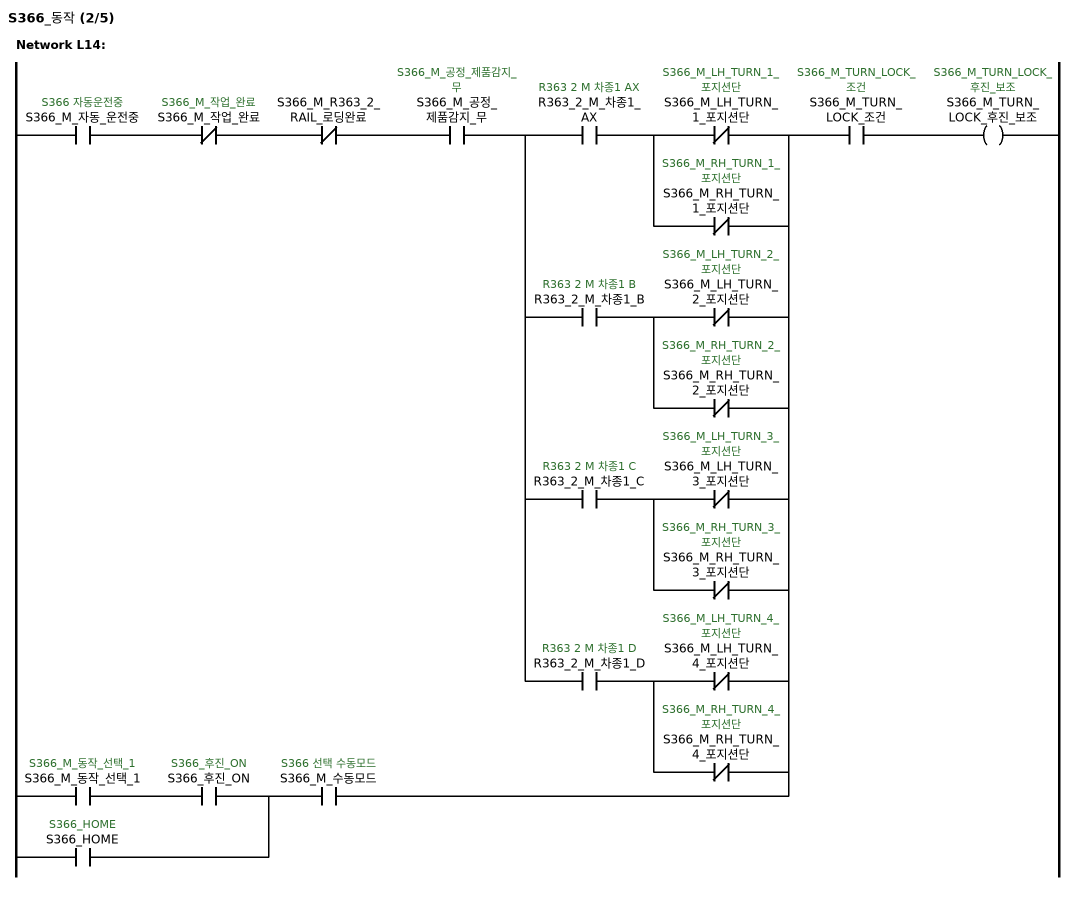
(* Rung L14 *)
S366_M_TURN_LOCK_후진_보조 := ((S366_M_자동_운전중 AND NOT S366_M_작업_완료 AND NOT S366_M_R363_2_RAIL_로딩완료 AND S366_M_공정_제품감지_무 AND ((R363_2_M_차종1_AX AND (NOT S366_M_LH_TURN_1_포지션단 OR NOT S366_M_RH_TURN_1_포지션단)) OR (R363_2_M_차종1_B AND (NOT S366_M_LH_TURN_2_포지션단 OR NOT S366_M_RH_TURN_2_포지션단)) OR (R363_2_M_차종1_C AND (NOT S366_M_LH_TURN_3_포지션단 OR NOT S366_M_RH_TURN_3_포지션단)) OR (R363_2_M_차종1_D AND (NOT S366_M_LH_TURN_4_포지션단 OR NOT S366_M_RH_TURN_4_포지션단)))) OR (((S366_M_동작_선택_1 AND S366_후진_ON) OR S366_HOME) AND S366_M_수동모드)) AND S366_M_TURN_LOCK_조건;

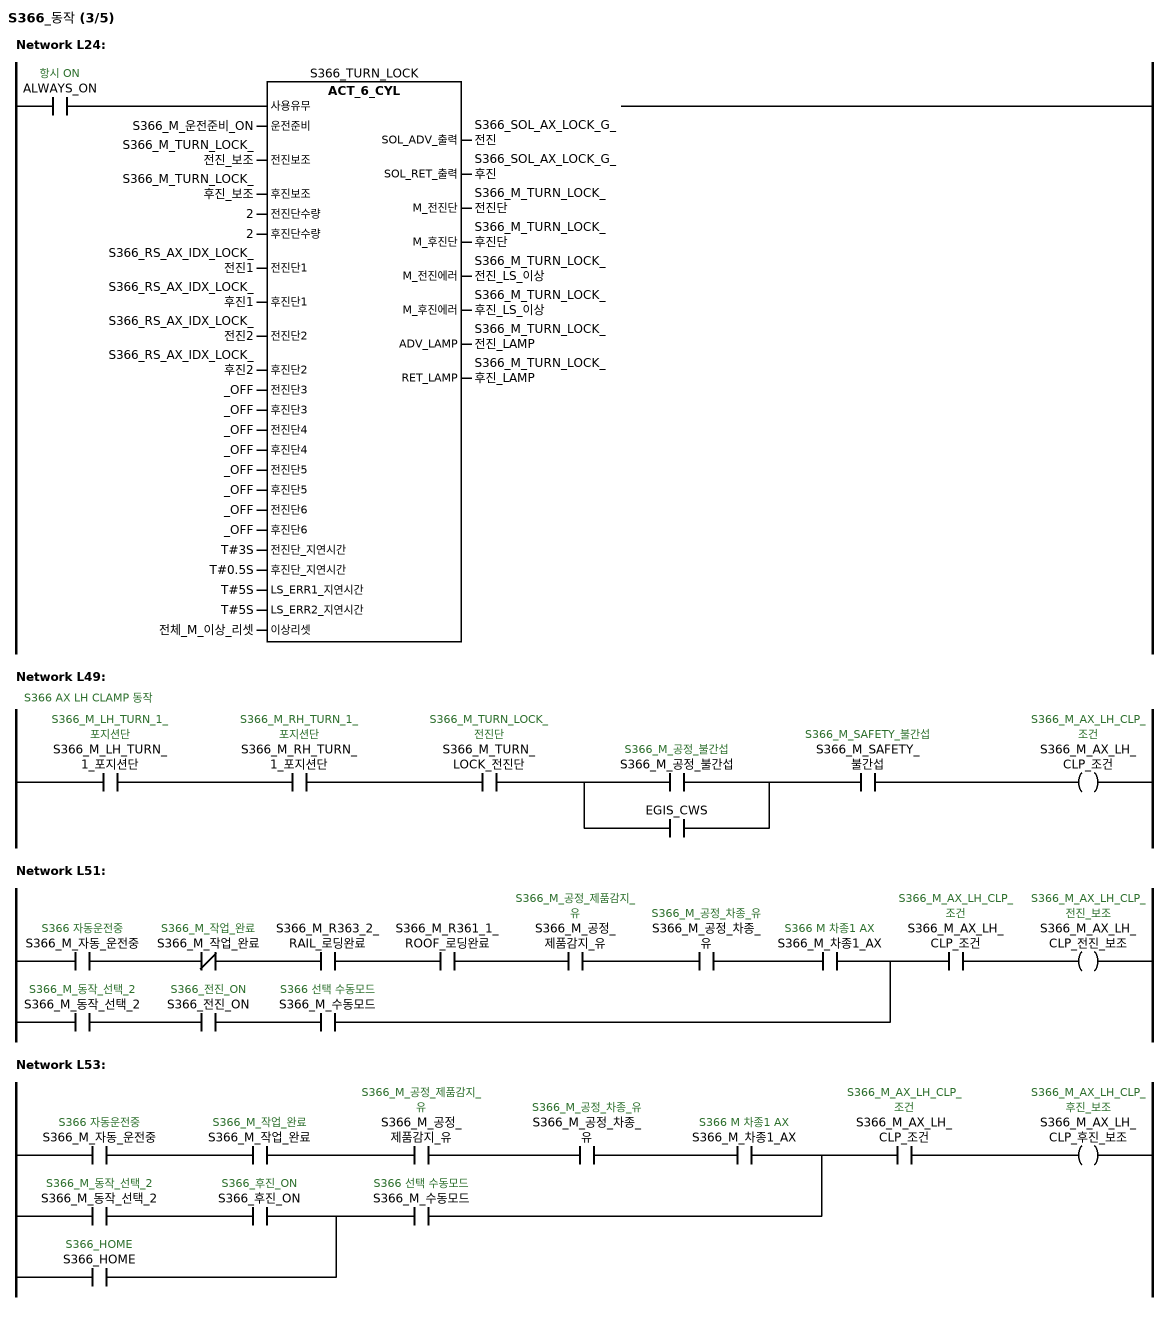
(* Rung L24 *)
S366_TURN_LOCK(사용유무 := ALWAYS_ON, 운전준비 := S366_M_운전준비_ON, 전진보조 := S366_M_TURN_LOCK_전진_보조, 후진보조 := S366_M_TURN_LOCK_후진_보조, 전진단수량 := 2, 후진단수량 := 2, 전진단1 := S366_RS_AX_IDX_LOCK_전진1, 후진단1 := S366_RS_AX_IDX_LOCK_후진1, 전진단2 := S366_RS_AX_IDX_LOCK_전진2, 후진단2 := S366_RS_AX_IDX_LOCK_후진2, 전진단3 := _OFF, 후진단3 := _OFF, 전진단4 := _OFF, 후진단4 := _OFF, 전진단5 := _OFF, 후진단5 := _OFF, 전진단6 := _OFF, 후진단6 := _OFF, 전진단_지연시간 := T#3S, 후진단_지연시간 := T#0.5S, LS_ERR1_지연시간 := T#5S, LS_ERR2_지연시간 := T#5S, 이상리셋 := 전체_M_이상_리셋, SOL_ADV_출력 => S366_SOL_AX_LOCK_G_전진, SOL_RET_출력 => S366_SOL_AX_LOCK_G_후진, M_전진단 => S366_M_TURN_LOCK_전진단, M_후진단 => S366_M_TURN_LOCK_후진단, M_전진에러 => S366_M_TURN_LOCK_전진_LS_이상, M_후진에러 => S366_M_TURN_LOCK_후진_LS_이상, ADV_LAMP => S366_M_TURN_LOCK_전진_LAMP, RET_LAMP => S366_M_TURN_LOCK_후진_LAMP);
(* S366 AX LH CLAMP 동작 *)
(* Rung L49 *)
S366_M_AX_LH_CLP_조건 := S366_M_LH_TURN_1_포지션단 AND S366_M_RH_TURN_1_포지션단 AND S366_M_TURN_LOCK_전진단 AND (S366_M_공정_불간섭 OR EGIS_CWS) AND S366_M_SAFETY_불간섭;
(* Rung L51 *)
S366_M_AX_LH_CLP_전진_보조 := ((S366_M_자동_운전중 AND NOT S366_M_작업_완료 AND S366_M_R363_2_RAIL_로딩완료 AND S366_M_R361_1_ROOF_로딩완료 AND S366_M_공정_제품감지_유 AND S366_M_공정_차종_유 AND S366_M_차종1_AX) OR (S366_M_동작_선택_2 AND S366_전진_ON AND S366_M_수동모드)) AND S366_M_AX_LH_CLP_조건;
(* Rung L53 *)
S366_M_AX_LH_CLP_후진_보조 := ((S366_M_자동_운전중 AND S366_M_작업_완료 AND S366_M_공정_제품감지_유 AND S366_M_공정_차종_유 AND S366_M_차종1_AX) OR (((S366_M_동작_선택_2 AND S366_후진_ON) OR S366_HOME) AND S366_M_수동모드)) AND S366_M_AX_LH_CLP_조건;

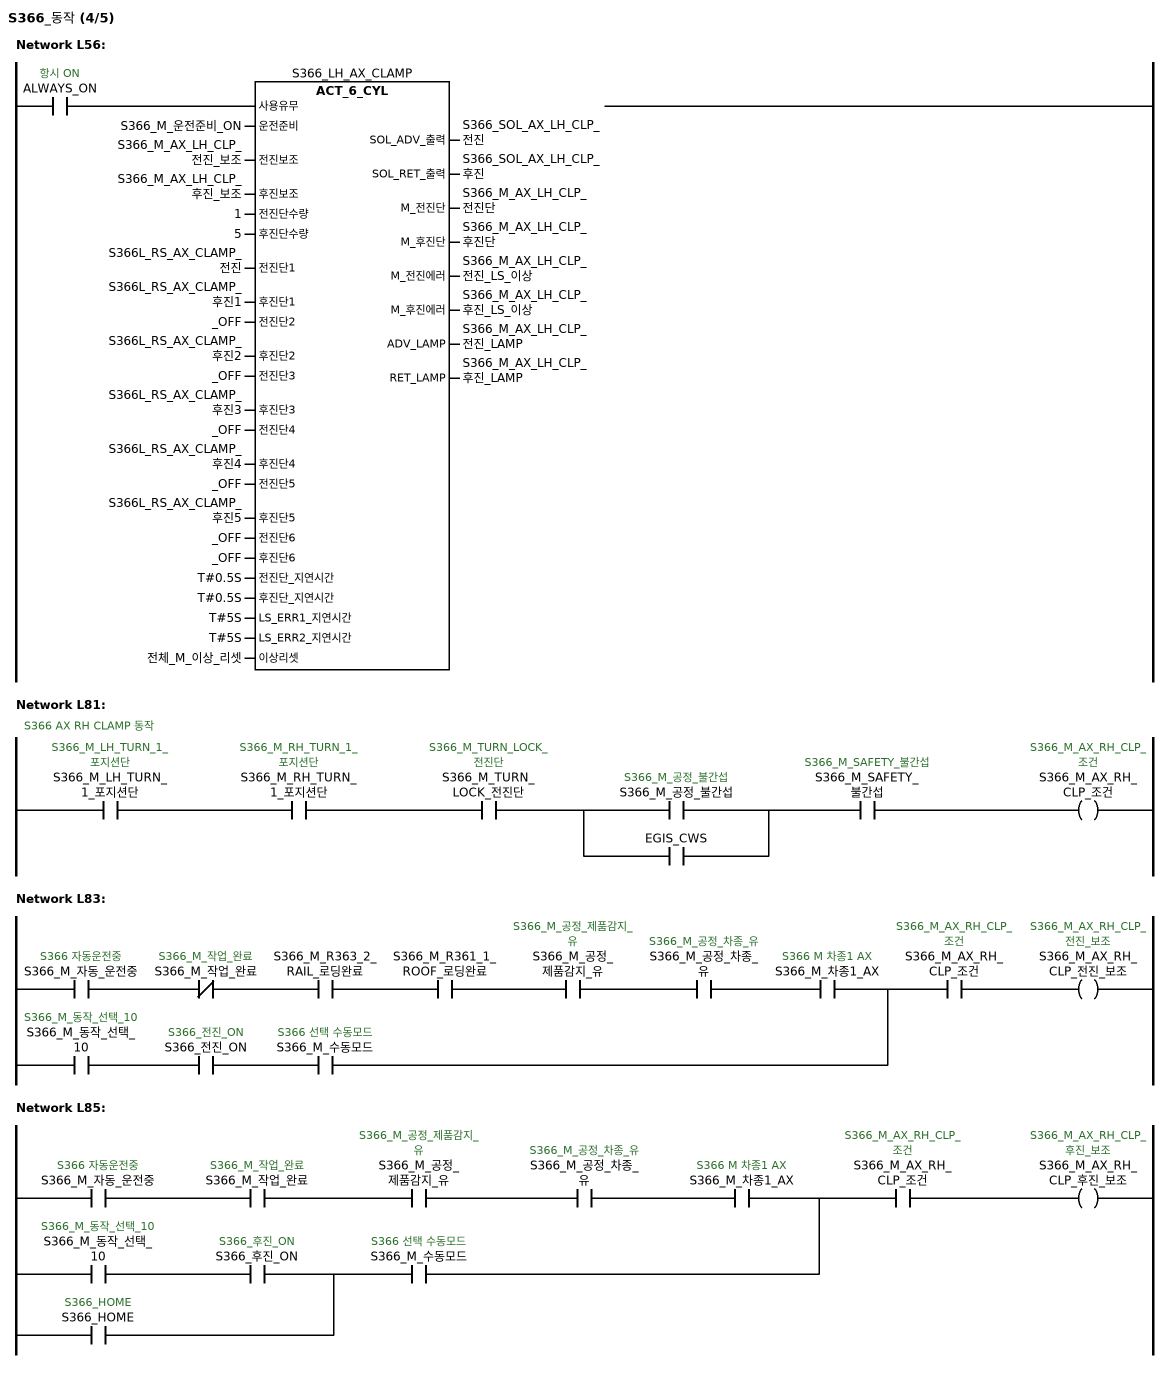
(* Rung L56 *)
S366_LH_AX_CLAMP(사용유무 := ALWAYS_ON, 운전준비 := S366_M_운전준비_ON, 전진보조 := S366_M_AX_LH_CLP_전진_보조, 후진보조 := S366_M_AX_LH_CLP_후진_보조, 전진단수량 := 1, 후진단수량 := 5, 전진단1 := S366L_RS_AX_CLAMP_전진, 후진단1 := S366L_RS_AX_CLAMP_후진1, 전진단2 := _OFF, 후진단2 := S366L_RS_AX_CLAMP_후진2, 전진단3 := _OFF, 후진단3 := S366L_RS_AX_CLAMP_후진3, 전진단4 := _OFF, 후진단4 := S366L_RS_AX_CLAMP_후진4, 전진단5 := _OFF, 후진단5 := S366L_RS_AX_CLAMP_후진5, 전진단6 := _OFF, 후진단6 := _OFF, 전진단_지연시간 := T#0.5S, 후진단_지연시간 := T#0.5S, LS_ERR1_지연시간 := T#5S, LS_ERR2_지연시간 := T#5S, 이상리셋 := 전체_M_이상_리셋, SOL_ADV_출력 => S366_SOL_AX_LH_CLP_전진, SOL_RET_출력 => S366_SOL_AX_LH_CLP_후진, M_전진단 => S366_M_AX_LH_CLP_전진단, M_후진단 => S366_M_AX_LH_CLP_후진단, M_전진에러 => S366_M_AX_LH_CLP_전진_LS_이상, M_후진에러 => S366_M_AX_LH_CLP_후진_LS_이상, ADV_LAMP => S366_M_AX_LH_CLP_전진_LAMP, RET_LAMP => S366_M_AX_LH_CLP_후진_LAMP);
(* S366 AX RH CLAMP 동작 *)
(* Rung L81 *)
S366_M_AX_RH_CLP_조건 := S366_M_LH_TURN_1_포지션단 AND S366_M_RH_TURN_1_포지션단 AND S366_M_TURN_LOCK_전진단 AND (S366_M_공정_불간섭 OR EGIS_CWS) AND S366_M_SAFETY_불간섭;
(* Rung L83 *)
S366_M_AX_RH_CLP_전진_보조 := ((S366_M_자동_운전중 AND NOT S366_M_작업_완료 AND S366_M_R363_2_RAIL_로딩완료 AND S366_M_R361_1_ROOF_로딩완료 AND S366_M_공정_제품감지_유 AND S366_M_공정_차종_유 AND S366_M_차종1_AX) OR (S366_M_동작_선택_10 AND S366_전진_ON AND S366_M_수동모드)) AND S366_M_AX_RH_CLP_조건;
(* Rung L85 *)
S366_M_AX_RH_CLP_후진_보조 := ((S366_M_자동_운전중 AND S366_M_작업_완료 AND S366_M_공정_제품감지_유 AND S366_M_공정_차종_유 AND S366_M_차종1_AX) OR (((S366_M_동작_선택_10 AND S366_후진_ON) OR S366_HOME) AND S366_M_수동모드)) AND S366_M_AX_RH_CLP_조건;

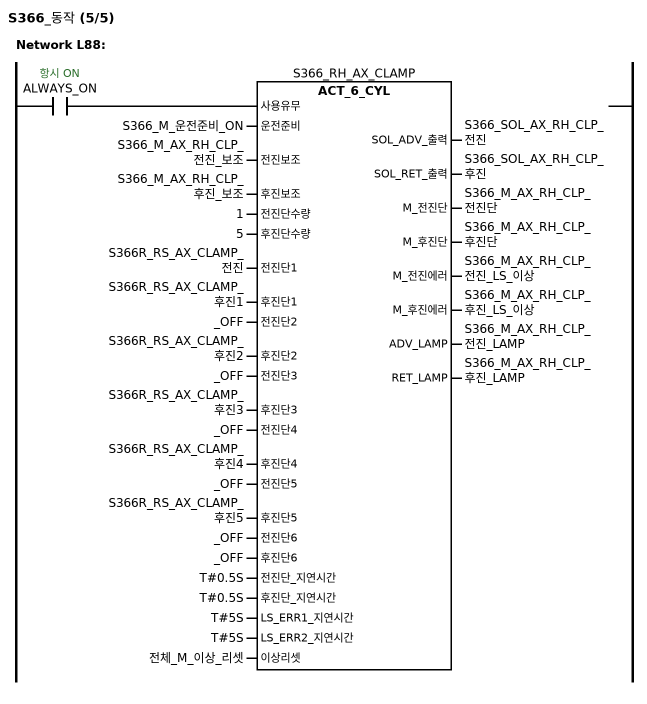
(* Rung L88 *)
S366_RH_AX_CLAMP(사용유무 := ALWAYS_ON, 운전준비 := S366_M_운전준비_ON, 전진보조 := S366_M_AX_RH_CLP_전진_보조, 후진보조 := S366_M_AX_RH_CLP_후진_보조, 전진단수량 := 1, 후진단수량 := 5, 전진단1 := S366R_RS_AX_CLAMP_전진, 후진단1 := S366R_RS_AX_CLAMP_후진1, 전진단2 := _OFF, 후진단2 := S366R_RS_AX_CLAMP_후진2, 전진단3 := _OFF, 후진단3 := S366R_RS_AX_CLAMP_후진3, 전진단4 := _OFF, 후진단4 := S366R_RS_AX_CLAMP_후진4, 전진단5 := _OFF, 후진단5 := S366R_RS_AX_CLAMP_후진5, 전진단6 := _OFF, 후진단6 := _OFF, 전진단_지연시간 := T#0.5S, 후진단_지연시간 := T#0.5S, LS_ERR1_지연시간 := T#5S, LS_ERR2_지연시간 := T#5S, 이상리셋 := 전체_M_이상_리셋, SOL_ADV_출력 => S366_SOL_AX_RH_CLP_전진, SOL_RET_출력 => S366_SOL_AX_RH_CLP_후진, M_전진단 => S366_M_AX_RH_CLP_전진단, M_후진단 => S366_M_AX_RH_CLP_후진단, M_전진에러 => S366_M_AX_RH_CLP_전진_LS_이상, M_후진에러 => S366_M_AX_RH_CLP_후진_LS_이상, ADV_LAMP => S366_M_AX_RH_CLP_전진_LAMP, RET_LAMP => S366_M_AX_RH_CLP_후진_LAMP);
END_PROGRAM

PROGRAM S366_외부설비(인덱스) (* task: 스캔 프로그램 *)
VAR
    A_차종 : BOOL;
    B_차종 : BOOL;
    C_차종 : BOOL;
    D_차종 : BOOL;
    INST1 : FB494_Robot_Hyundai_HMMI_v1;
    R366_1_M_RB_PROG_NO : INT;
    T366_LH_TURN_LS_이상 : TON;
    T366_LH_TURN_POSI_1 : TON;
    T366_LH_TURN_POSI_2 : TON;
    T366_LH_TURN_POSI_3 : TON;
    T366_LH_TURN_POSI_4 : TON;
    T366_RH_TURN_LS_이상 : TON;
    T366_RH_TURN_POSI_5 : TON;
    T366_RH_TURN_POSI_6 : TON;
    T366_RH_TURN_POSI_7 : TON;
    T366_RH_TURN_POSI_8 : TON;
    로보트제외 : BOOL;
END_VAR
VAR_EXTERNAL
    EGIS_CWS : BOOL;
    MCP_PBL_운전준비_ON : BOOL; (* AT %MW87630.0 *) (* MCP_PBL_운전준비_ON *)
    R366_1_I_RB_INPUT : ARRAY[0..3] OF WORD; (* AT %MW84060 *) (* R366_1_I_RB_INPUT *)
    R366_1_M_I_RB_1차_작업완료 : BOOL; (* AT %MW20061.2 *) (* R366_1_M_I_RB_1차_작업완료 *)
    R366_1_M_I_RB_2차_작업완료 : BOOL; (* AT %MW20061.3 *) (* R366_1_M_I_RB_2차_작업완료 *)
    R366_1_M_I_RB_3차_작업완료 : BOOL; (* AT %MW20061.4 *) (* R366_1_M_I_RB_3차_작업완료 *)
    R366_1_M_I_RB_4차_작업완료 : BOOL; (* AT %MW20061.5 *) (* R366_1_M_I_RB_4차_작업완료 *)
    R366_1_M_I_RB_5차_작업완료 : BOOL; (* AT %MW20061.6 *) (* R366_1_M_I_RB_5차_작업완료 *)
    R366_1_M_I_RB_6차_작업완료 : BOOL; (* AT %MW20061.7 *) (* R366_1_M_I_RB_6차_작업완료 *)
    R366_1_M_I_RB_7차_작업완료 : BOOL; (* AT %MW20061.8 *) (* R366_1_M_I_RB_7차_작업완료 *)
    R366_1_M_I_RB_PAUSE_보조 : BOOL; (* AT %MW20060.5 *) (* R366_1_M_I_RB_PAUSE_보조 *)
    R366_1_M_I_RB_PLC_RUN_CHK_이상 : BOOL; (* AT %MW20060.7 *) (* R366_1_M_I_RB_PLC_RUN_CHK_이상 *)
    R366_1_M_I_RB_간섭무_1 : BOOL; (* AT %MW20062.0 *) (* R366_1_M_I_RB_간섭무_1 *)
    R366_1_M_I_RB_간섭무_10 : BOOL; (* AT %MW20062.9 *) (* R366_1_M_I_RB_간섭무_10 *)
    R366_1_M_I_RB_간섭무_11 : BOOL; (* AT %MW20062.10 *) (* R366_1_M_I_RB_간섭무_11 *)
    R366_1_M_I_RB_간섭무_12 : BOOL; (* AT %MW20062.11 *) (* R366_1_M_I_RB_간섭무_12 *)
    R366_1_M_I_RB_간섭무_2 : BOOL; (* AT %MW20062.1 *) (* R366_1_M_I_RB_간섭무_2 *)
    R366_1_M_I_RB_간섭무_3 : BOOL; (* AT %MW20062.2 *) (* R366_1_M_I_RB_간섭무_3 *)
    R366_1_M_I_RB_간섭무_4 : BOOL; (* AT %MW20062.3 *) (* R366_1_M_I_RB_간섭무_4 *)
    R366_1_M_I_RB_간섭무_5 : BOOL; (* AT %MW20062.4 *) (* R366_1_M_I_RB_간섭무_5 *)
    R366_1_M_I_RB_간섭무_6 : BOOL; (* AT %MW20062.5 *) (* R366_1_M_I_RB_간섭무_6 *)
    R366_1_M_I_RB_간섭무_7 : BOOL; (* AT %MW20062.6 *) (* R366_1_M_I_RB_간섭무_7 *)
    R366_1_M_I_RB_간섭무_8 : BOOL; (* AT %MW20062.7 *) (* R366_1_M_I_RB_간섭무_8 *)
    R366_1_M_I_RB_간섭무_9 : BOOL; (* AT %MW20062.8 *) (* R366_1_M_I_RB_간섭무_9 *)
    R366_1_M_I_RB_비상정지 : BOOL; (* AT %MW20060.4 *) (* R366_1_M_I_RB_비상정지 *)
    R366_1_M_I_RB_운전준비 : BOOL; (* AT %MW20060.0 *) (* R366_1_M_I_RB_운전준비 *)
    R366_1_M_I_RB_원위치 : BOOL; (* AT %MW20060.3 *) (* R366_1_M_I_RB_원위치 *)
    R366_1_M_I_RB_이상 : BOOL; (* AT %MW20060.2 *) (* R366_1_M_I_RB_이상 *)
    R366_1_M_I_RB_자동 : BOOL; (* AT %MW20060.1 *) (* R366_1_M_I_RB_자동 *)
    R366_1_M_I_RB_최종작업완료 : BOOL; (* AT %MW20061.0 *) (* R366_1_M_I_RB_최종작업완료 *)
    R366_1_M_I_RB_프로그램_이상 : BOOL; (* AT %MW20060.6 *) (* R366_1_M_I_RB_프로그램_이상 *)
    R366_1_M_O_RB_1_CYCLE_SET : BOOL; (* AT %MW21060.3 *) (* R366_1_M_O_RB_1_CYCLE_SET *)
    R366_1_M_O_RB_1차_작업완료_리셋 : BOOL; (* AT %MW21062.0 *) (* R366_1_M_O_RB_1차_작업완료_리셋 *)
    R366_1_M_O_RB_2차_작업완료_리셋 : BOOL; (* AT %MW21062.1 *) (* R366_1_M_O_RB_2차_작업완료_리셋 *)
    R366_1_M_O_RB_2차_진입OK : BOOL; (* AT %MW21061.8 *) (* R366_1_M_O_RB_2차_진입OK *)
    R366_1_M_O_RB_3차_작업완료_리셋 : BOOL; (* AT %MW21062.2 *) (* R366_1_M_O_RB_3차_작업완료_리셋 *)
    R366_1_M_O_RB_3차_진입OK : BOOL; (* AT %MW21061.9 *) (* R366_1_M_O_RB_3차_진입OK *)
    R366_1_M_O_RB_4차_작업완료_리셋 : BOOL; (* AT %MW21062.3 *) (* R366_1_M_O_RB_4차_작업완료_리셋 *)
    R366_1_M_O_RB_4차_진입OK : BOOL; (* AT %MW21061.10 *) (* R366_1_M_O_RB_4차_진입OK *)
    R366_1_M_O_RB_5차_작업완료_리셋 : BOOL; (* AT %MW21062.4 *) (* R366_1_M_O_RB_5차_작업완료_리셋 *)
    R366_1_M_O_RB_5차_진입OK : BOOL; (* AT %MW21061.11 *) (* R366_1_M_O_RB_5차_진입OK *)
    R366_1_M_O_RB_6차_작업완료_리셋 : BOOL; (* AT %MW21062.5 *) (* R366_1_M_O_RB_6차_작업완료_리셋 *)
    R366_1_M_O_RB_6차_진입OK : BOOL; (* AT %MW21061.12 *) (* R366_1_M_O_RB_6차_진입OK *)
    R366_1_M_O_RB_7차_작업완료_리셋 : BOOL; (* AT %MW21062.6 *) (* R366_1_M_O_RB_7차_작업완료_리셋 *)
    R366_1_M_O_RB_7차_진입OK : BOOL; (* AT %MW21061.13 *) (* R366_1_M_O_RB_7차_진입OK *)
    R366_1_M_O_RB_ATD_OK : BOOL; (* AT %MW21060.6 *) (* R366_1_M_O_RB_ATD_OK *)
    R366_1_M_O_RB_PLT_10_진입OK : BOOL; (* AT %MW21063.10 *) (* R366_1_M_O_RB_PLT_10_진입OK *)
    R366_1_M_O_RB_PLT_11_진입OK : BOOL; (* AT %MW21063.11 *) (* R366_1_M_O_RB_PLT_11_진입OK *)
    R366_1_M_O_RB_PLT_12_진입OK : BOOL; (* AT %MW21063.12 *) (* R366_1_M_O_RB_PLT_12_진입OK *)
    R366_1_M_O_RB_PLT_1_진입OK : BOOL; (* AT %MW21063.1 *) (* R366_1_M_O_RB_PLT_1_진입OK *)
    R366_1_M_O_RB_PLT_2_진입OK : BOOL; (* AT %MW21063.2 *) (* R366_1_M_O_RB_PLT_2_진입OK *)
    R366_1_M_O_RB_PLT_3_진입OK : BOOL; (* AT %MW21063.3 *) (* R366_1_M_O_RB_PLT_3_진입OK *)
    R366_1_M_O_RB_PLT_4_진입OK : BOOL; (* AT %MW21063.4 *) (* R366_1_M_O_RB_PLT_4_진입OK *)
    R366_1_M_O_RB_PLT_5_진입OK : BOOL; (* AT %MW21063.5 *) (* R366_1_M_O_RB_PLT_5_진입OK *)
    R366_1_M_O_RB_PLT_6_진입OK : BOOL; (* AT %MW21063.6 *) (* R366_1_M_O_RB_PLT_6_진입OK *)
    R366_1_M_O_RB_PLT_7_진입OK : BOOL; (* AT %MW21063.7 *) (* R366_1_M_O_RB_PLT_7_진입OK *)
    R366_1_M_O_RB_PLT_8_진입OK : BOOL; (* AT %MW21063.8 *) (* R366_1_M_O_RB_PLT_8_진입OK *)
    R366_1_M_O_RB_PLT_9_진입OK : BOOL; (* AT %MW21063.9 *) (* R366_1_M_O_RB_PLT_9_진입OK *)
    R366_1_M_O_RB_PLT_카운터리셋_보조 : BOOL; (* AT %MW21060.10 *) (* R366_1_M_O_RB_PLT_카운터리셋_보조 *)
    R366_1_M_O_RB_RESTART_OK : BOOL; (* AT %MW21060.2 *) (* R366_1_M_O_RB_RESTART_OK *)
    R366_1_M_O_RB_START_OK : BOOL; (* AT %MW21060.0 *) (* R366_1_M_O_RB_START_OK *)
    R366_1_M_O_RB_TEST_MODE_5000회 : BOOL; (* AT %MW21060.12 *) (* R366_1_M_O_RB_TEST_MODE_5000회 *)
    R366_1_M_O_RB_TIP_교체_시작 : BOOL; (* AT %MW21060.7 *) (* R366_1_M_O_RB_TIP_교체_시작 *)
    R366_1_M_O_RB_TIP_교체_완료 : BOOL; (* AT %MW21060.8 *) (* R366_1_M_O_RB_TIP_교체_완료 *)
    R366_1_M_O_RB_VIP_MODE : BOOL; (* AT %MW21060.11 *) (* R366_1_M_O_RB_VIP_MODE *)
    R366_1_M_O_RB_냉각수_차단_요청 : BOOL; (* AT %MW21060.9 *) (* R366_1_M_O_RB_냉각수_차단_요청 *)
    R366_1_M_O_RB_진입OK_AX차종 : BOOL; (* AT %MW21061.0 *) (* R366_1_M_O_RB_진입OK_AX차종 *)
    R366_1_M_O_RB_진입OK_B차종 : BOOL; (* AT %MW21061.1 *) (* R366_1_M_O_RB_진입OK_B차종 *)
    R366_1_M_O_RB_진입OK_C차종 : BOOL; (* AT %MW21061.2 *) (* R366_1_M_O_RB_진입OK_C차종 *)
    R366_1_M_O_RB_진입OK_D차종 : BOOL; (* AT %MW21061.3 *) (* R366_1_M_O_RB_진입OK_D차종 *)
    R366_1_M_O_RB_진입OK_E차종 : BOOL; (* AT %MW21061.4 *) (* R366_1_M_O_RB_진입OK_E차종 *)
    R366_1_M_O_RB_진입OK_F차종 : BOOL; (* AT %MW21061.5 *) (* R366_1_M_O_RB_진입OK_F차종 *)
    R366_1_M_O_RB_진입OK_G차종 : BOOL; (* AT %MW21061.6 *) (* R366_1_M_O_RB_진입OK_G차종 *)
    R366_1_M_O_RB_진입OK_H차종 : BOOL; (* AT %MW21061.7 *) (* R366_1_M_O_RB_진입OK_H차종 *)
    R366_1_M_O_RB_최종_작업완료_리셋 : BOOL; (* AT %MW21060.5 *) (* R366_1_M_O_RB_최종_작업완료_리셋 *)
    R366_1_M_O_RB_프로그램_OK : BOOL; (* AT %MW21060.1 *) (* R366_1_M_O_RB_프로그램_OK *)
    R366_1_O_RB_OUTPUT : ARRAY[0..3] OF WORD; (* AT %MW94060 *) (* R366_1_O_RB_OUTPUT *)
    S362_6_INV3_BRAKE_CR_ON : BOOL; (* AT %MW95015.7 *) (* S362_6_INV3_BRAKE_CR_ON *)
    S362_6_INV3_RETURN : BOOL; (* AT %MW95015.1 *) (* S362_6_INV3_RETURN *)
    S362_6_INV3_TURN : BOOL; (* AT %MW95015.0 *) (* S362_6_INV3_TURN *)
    S362_6_INV4_BRAKE_CR_ON : BOOL; (* AT %MW95015.15 *) (* S362_6_INV4_BRAKE_CR_ON *)
    S362_6_INV4_RETURN : BOOL; (* AT %MW95015.9 *) (* S362_6_INV4_RETURN *)
    S362_6_INV4_TURN : BOOL; (* AT %MW95015.8 *) (* S362_6_INV4_TURN *)
    S366_INDEX_LH_TURN_감지1 : BOOL; (* AT %MW86101.4 *) (* S366_INDEX_LH_TURN_감지1 *)
    S366_INDEX_LH_TURN_감지2 : BOOL; (* AT %MW86101.5 *) (* S366_INDEX_LH_TURN_감지2 *)
    S366_INDEX_LH_TURN_감지3 : BOOL; (* AT %MW86101.6 *) (* S366_INDEX_LH_TURN_감지3 *)
    S366_INDEX_LH_TURN_원점 : BOOL; (* AT %MW86101.7 *) (* S366_INDEX_LH_TURN_원점 *)
    S366_INDEX_RH_TURN_감지1 : BOOL; (* AT %MW86101.0 *) (* S366_INDEX_RH_TURN_감지1 *)
    S366_INDEX_RH_TURN_감지2 : BOOL; (* AT %MW86101.1 *) (* S366_INDEX_RH_TURN_감지2 *)
    S366_INDEX_RH_TURN_감지3 : BOOL; (* AT %MW86101.2 *) (* S366_INDEX_RH_TURN_감지3 *)
    S366_INDEX_RH_TURN_원점 : BOOL; (* AT %MW86101.3 *) (* S366_INDEX_RH_TURN_원점 *)
END_VAR
VAR_EXTERNAL RETAIN
    MCP_M_부저_정지 : BOOL; (* AT %MW350.5 *) (* MCP 부저정지 *)
    MCP_M_비상정지 : BOOL; (* AT %MW350.7 *) (* MCP 비상정지 이상 *)
    R363_2_M_차종1_AX : BOOL; (* AT %MW10041.0 *) (* R363 2 M 차종1 AX *)
    R363_2_M_차종1_B : BOOL; (* AT %MW10041.1 *) (* R363 2 M 차종1 B *)
    R363_2_M_차종1_C : BOOL; (* AT %MW10041.2 *) (* R363 2 M 차종1 C *)
    R363_2_M_차종1_D : BOOL; (* AT %MW10041.3 *) (* R363 2 M 차종1 D *)
    R363_2_M_차종_유 : BOOL; (* AT %MW1002.2 *) (* S362_M_공정_차종_보조 *)
    S362_M_공정_제품감지_무 : BOOL; (* AT %MW1001.5 *) (* S362_M_공정_제품감지_무 *)
    S366_M_AX_LH_CLP_후진단 : BOOL; (* AT %MW3104.4 *) (* S366_M_AX_LH_CLP_후진단 *)
    S366_M_AX_RH_CLP_후진단 : BOOL; (* AT %MW3112.4 *) (* S366_M_AX_RH_CLP_후진단 *)
    S366_M_LH_STEP_MOVE_리셋_PLS : BOOL; (* AT %MW3101.14 *) (* S366_M_LH_STEP_MOVE_리셋_PLS *)
    S366_M_LH_TURN_1_포지션단 : BOOL; (* AT %MW3101.3 *) (* S366_M_LH_TURN_1_포지션단 *)
    S366_M_LH_TURN_2_포지션단 : BOOL; (* AT %MW3101.4 *) (* S366_M_LH_TURN_2_포지션단 *)
    S366_M_LH_TURN_3_포지션단 : BOOL; (* AT %MW3101.5 *) (* S366_M_LH_TURN_3_포지션단 *)
    S366_M_LH_TURN_4_포지션단 : BOOL; (* AT %MW3101.6 *) (* S366_M_LH_TURN_4_포지션단 *)
    S366_M_LH_TURN_LS_이상 : BOOL; (* AT %MW3101.7 *) (* S366_M_LH_TURN_LS_이상 *)
    S366_M_LH_TURN_MOVE_완료 : BOOL; (* AT %MW3101.8 *) (* S366_M_LH_TURN_MOVE_완료 *)
    S366_M_LH_TURN_수동_STEP_전진_보조 : BOOL; (* AT %MW3101.11 *) (* S366_M_LH_TURN_수동_STEP_전진_보조 *)
    S366_M_LH_TURN_수동_STEP_후진_보조 : BOOL; (* AT %MW3101.12 *) (* S366_M_LH_TURN_수동_STEP_후진_보조 *)
    S366_M_LH_TURN_수동_전진_보조 : BOOL; (* AT %MW3101.9 *) (* S366_M_LH_TURN_수동_전진_보조 *)
    S366_M_LH_TURN_수동_후진_보조 : BOOL; (* AT %MW3101.10 *) (* S366_M_LH_TURN_수동_후진_보조 *)
    S366_M_LH_TURN_전진_보조 : BOOL; (* AT %MW3101.1 *) (* S366_M_LH_TURN_전진_보조 *)
    S366_M_LH_TURN_조건 : BOOL; (* AT %MW3101.0 *) (* S366_M_LH_TURN_조건 *)
    S366_M_LH_TURN_후진_보조 : BOOL; (* AT %MW3101.2 *) (* S366_M_LH_TURN_후진_보조 *)
    S366_M_LH_자동_MOVE_리셋_PLS : BOOL; (* AT %MW3101.13 *) (* S366_M_LH_자동_MOVE_리셋_PLS *)
    S366_M_R363_2_RAIL_로딩완료 : BOOL; (* AT %MW3001.1 *)
    S366_M_RH_STEP_MOVE_리셋_PLS : BOOL; (* AT %MW3109.14 *) (* S366_M_RH_STEP_MOVE_리셋_PLS *)
    S366_M_RH_TURN_1_포지션단 : BOOL; (* AT %MW3109.3 *) (* S366_M_RH_TURN_1_포지션단 *)
    S366_M_RH_TURN_2_포지션단 : BOOL; (* AT %MW3109.4 *) (* S366_M_RH_TURN_2_포지션단 *)
    S366_M_RH_TURN_3_포지션단 : BOOL; (* AT %MW3109.5 *) (* S366_M_RH_TURN_3_포지션단 *)
    S366_M_RH_TURN_4_포지션단 : BOOL; (* AT %MW3109.6 *) (* S366_M_RH_TURN_4_포지션단 *)
    S366_M_RH_TURN_LS_이상 : BOOL; (* AT %MW3109.7 *) (* S366_M_RH_TURN_LS_이상 *)
    S366_M_RH_TURN_MOVE_완료 : BOOL; (* AT %MW3109.8 *) (* S366_M_RH_TURN_MOVE_완료 *)
    S366_M_RH_TURN_수동_STEP_전진_보조 : BOOL; (* AT %MW3109.11 *) (* S366_M_RH_TURN_수동_STEP_전진_보조 *)
    S366_M_RH_TURN_수동_STEP_후진_보조 : BOOL; (* AT %MW3109.12 *) (* S366_M_RH_TURN_수동_STEP_후진_보조 *)
    S366_M_RH_TURN_수동_전진_보조 : BOOL; (* AT %MW3109.9 *) (* S366_M_RH_TURN_수동_전진_보조 *)
    S366_M_RH_TURN_수동_후진_보조 : BOOL; (* AT %MW3109.10 *) (* S366_M_RH_TURN_수동_후진_보조 *)
    S366_M_RH_TURN_전진_보조 : BOOL; (* AT %MW3109.1 *) (* S366_M_RH_TURN_전진_보조 *)
    S366_M_RH_TURN_조건 : BOOL; (* AT %MW3109.0 *) (* S366_M_RH_TURN_조건 *)
    S366_M_RH_TURN_후진_보조 : BOOL; (* AT %MW3109.2 *) (* S366_M_RH_TURN_후진_보조 *)
    S366_M_RH_자동_MOVE_리셋_PLS : BOOL; (* AT %MW3109.13 *) (* S366_M_RH_자동_MOVE_리셋_PLS *)
    S366_M_SAFETY_불간섭 : BOOL; (* AT %MW3004.4 *) (* S366_M_SAFETY_불간섭 *)
    S366_M_TURN_LOCK_후진단 : BOOL; (* AT %MW3100.4 *) (* S366_M_TURN_LOCK_후진단 *)
    S366_M_공정_불간섭 : BOOL; (* AT %MW3004.1 *) (* S366_M_공정_불간섭 *)
    S366_M_공정_제품감지_무 : BOOL; (* AT %MW3001.7 *) (* S366_M_공정_제품감지_무 *)
    S366_M_공정_차종_AX : BOOL; (* AT %MW3002.3 *) (* S366_M_공정_차종_AX *)
    S366_M_동작_선택_13 : BOOL; (* AT %MW3040.12 *) (* S366_M_동작_선택_13 *)
    S366_M_동작_선택_14 : BOOL; (* AT %MW3040.13 *) (* S366_M_동작_선택_14 *)
    S366_M_동작_선택_15 : BOOL; (* AT %MW3040.14 *) (* S366_M_동작_선택_15 *)
    S366_M_동작_선택_16 : BOOL; (* AT %MW3040.15 *) (* S366_M_동작_선택_16 *)
    S366_M_동작_선택_5 : BOOL; (* AT %MW3040.4 *) (* S366_M_동작_선택_5 *)
    S366_M_동작_선택_6 : BOOL; (* AT %MW3040.5 *) (* S366_M_동작_선택_6 *)
    S366_M_동작_선택_7 : BOOL; (* AT %MW3040.6 *) (* S366_M_동작_선택_7 *)
    S366_M_동작_선택_8 : BOOL; (* AT %MW3040.7 *) (* S366_M_동작_선택_8 *)
    S366_M_수동모드 : BOOL; (* AT %MW3000.3 *) (* S366 선택 수동모드 *)
    S366_M_운전준비_ON : BOOL; (* AT %MW3000.0 *) (* S366 운전준비 ON *)
    S366_M_자동_START : BOOL; (* AT %MW3000.5 *) (* S366 자동운전중 *)
    S366_M_자동_운전중 : BOOL; (* AT %MW3000.4 *) (* S366 자동운전중 *)
    S366_M_작업_완료 : BOOL; (* AT %MW3001.0 *) (* S366_M_작업_완료 *)
    S366_M_총괄_이상 : BOOL; (* AT %MW3009.0 *) (* S366_M_총괄_이상 *)
    S366_전진_ON : BOOL; (* AT %MW3048.1 *) (* S366_전진_ON *)
    S366_후진_ON : BOOL; (* AT %MW3048.2 *) (* S366_후진_ON *)
    전체_M_이상_리셋 : BOOL; (* AT %MW308.2 *) (* ALL공정 PB 이상리셋 *)
END_VAR
VAR
    _e1 : R_TRIG;
    _e2 : R_TRIG;
    _e3 : R_TRIG;
    _e4 : R_TRIG;
END_VAR

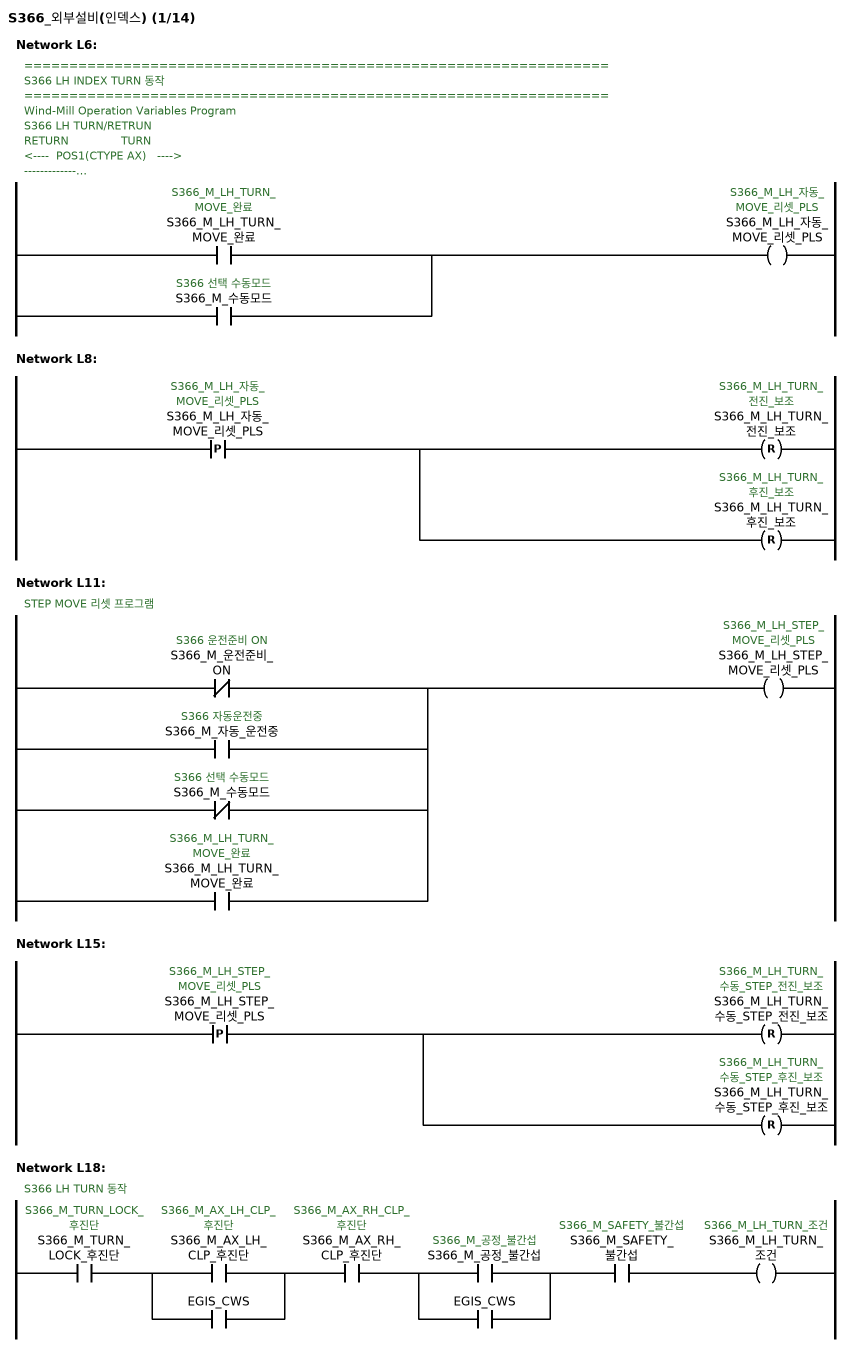
(* ================================================================= *)
(* S366 LH INDEX TURN 동작 *)
(* ================================================================= *)
(* Wind-Mill Operation Variables Program / S366 LH TURN/RETRUN *)
(* RETURN               TURN / <----  POS1(CTYPE AX)   ----> / -------------- / l              l / l              l / l              l / POS2 (CTYPE B) l              l  POS4 (CTYPE D) / l              l / l              l / l              l / -------------- / POS3 (CTYPE C) *)
(* 자동 MOVE 리셋 프로그램 *)
(* Rung L6 *)
S366_M_LH_자동_MOVE_리셋_PLS := S366_M_LH_TURN_MOVE_완료 OR S366_M_수동모드;
(* Rung L8 *)
_e1(CLK := S366_M_LH_자동_MOVE_리셋_PLS);
IF _e1.Q THEN
    S366_M_LH_TURN_전진_보조 := FALSE;
    S366_M_LH_TURN_후진_보조 := FALSE;
END_IF;
(* STEP MOVE 리셋 프로그램 *)
(* Rung L11 *)
S366_M_LH_STEP_MOVE_리셋_PLS := NOT S366_M_운전준비_ON OR S366_M_자동_운전중 OR NOT S366_M_수동모드 OR S366_M_LH_TURN_MOVE_완료;
(* Rung L15 *)
_e2(CLK := S366_M_LH_STEP_MOVE_리셋_PLS);
IF _e2.Q THEN
    S366_M_LH_TURN_수동_STEP_전진_보조 := FALSE;
    S366_M_LH_TURN_수동_STEP_후진_보조 := FALSE;
END_IF;
(* S366 LH TURN 동작 *)
(* Rung L18 *)
S366_M_LH_TURN_조건 := S366_M_TURN_LOCK_후진단 AND (S366_M_AX_LH_CLP_후진단 OR EGIS_CWS) AND S366_M_AX_RH_CLP_후진단 AND (S366_M_공정_불간섭 OR EGIS_CWS) AND S366_M_SAFETY_불간섭;

